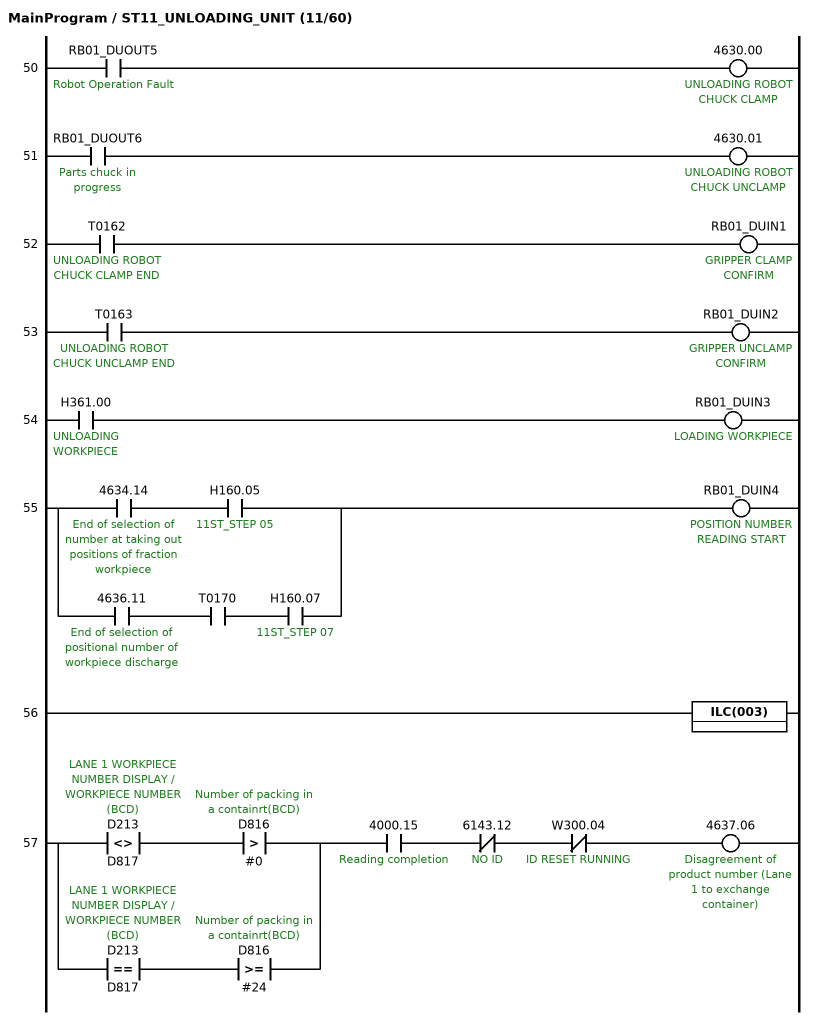
; [picture p528: MainProgram / ST11_UNLOADING_UNIT, rungs 50-57]
; rung 50
LD RB01_DUOUT5  ; Robot Operation Fault
OUT 4630.00  ; UNLOADING ROBOT CHUCK CLAMP
; rung 51
LD RB01_DUOUT6  ; Parts chuck in progress
OUT 4630.01  ; UNLOADING ROBOT CHUCK UNCLAMP
; rung 52
LD T0162  ; UNLOADING ROBOT CHUCK CLAMP END
OUT RB01_DUIN1  ; GRIPPER CLAMP CONFIRM
; rung 53
LD T0163  ; UNLOADING ROBOT CHUCK UNCLAMP END
OUT RB01_DUIN2  ; GRIPPER UNCLAMP CONFIRM
; rung 54
LD H361.00  ; UNLOADING WORKPIECE
OUT RB01_DUIN3  ; LOADING WORKPIECE
; rung 55
LD 4634.14  ; End of selection of number at taking out positions of fraction workpiece
AND H160.05  ; 11ST_STEP 05
LD 4636.11  ; End of selection of positional number of workpiece discharge
AND T0170
AND H160.07  ; 11ST_STEP 07
ORLD
OUT RB01_DUIN4  ; POSITION NUMBER READING START
; rung 56
ILC(003)
; rung 57
LD<>(305) D213 D817  ; LANE 1 WORKPIECE NUMBER DISPLAY, WORKPIECE NUMBER (BCD)
AND>(320) D816 #0  ; Number of packing in a containrt(BCD)
LD=(300) D213 D817  ; LANE 1 WORKPIECE NUMBER DISPLAY, WORKPIECE NUMBER (BCD)
AND>=(325) D816 #24  ; Number of packing in a containrt(BCD)
ORLD
AND 4000.15  ; Reading completion
ANDNOT 6143.12  ; NO ID
ANDNOT W300.04  ; ID RESET RUNNING
OUT 4637.06  ; Disagreement of product number (Lane 1 to exchange container)

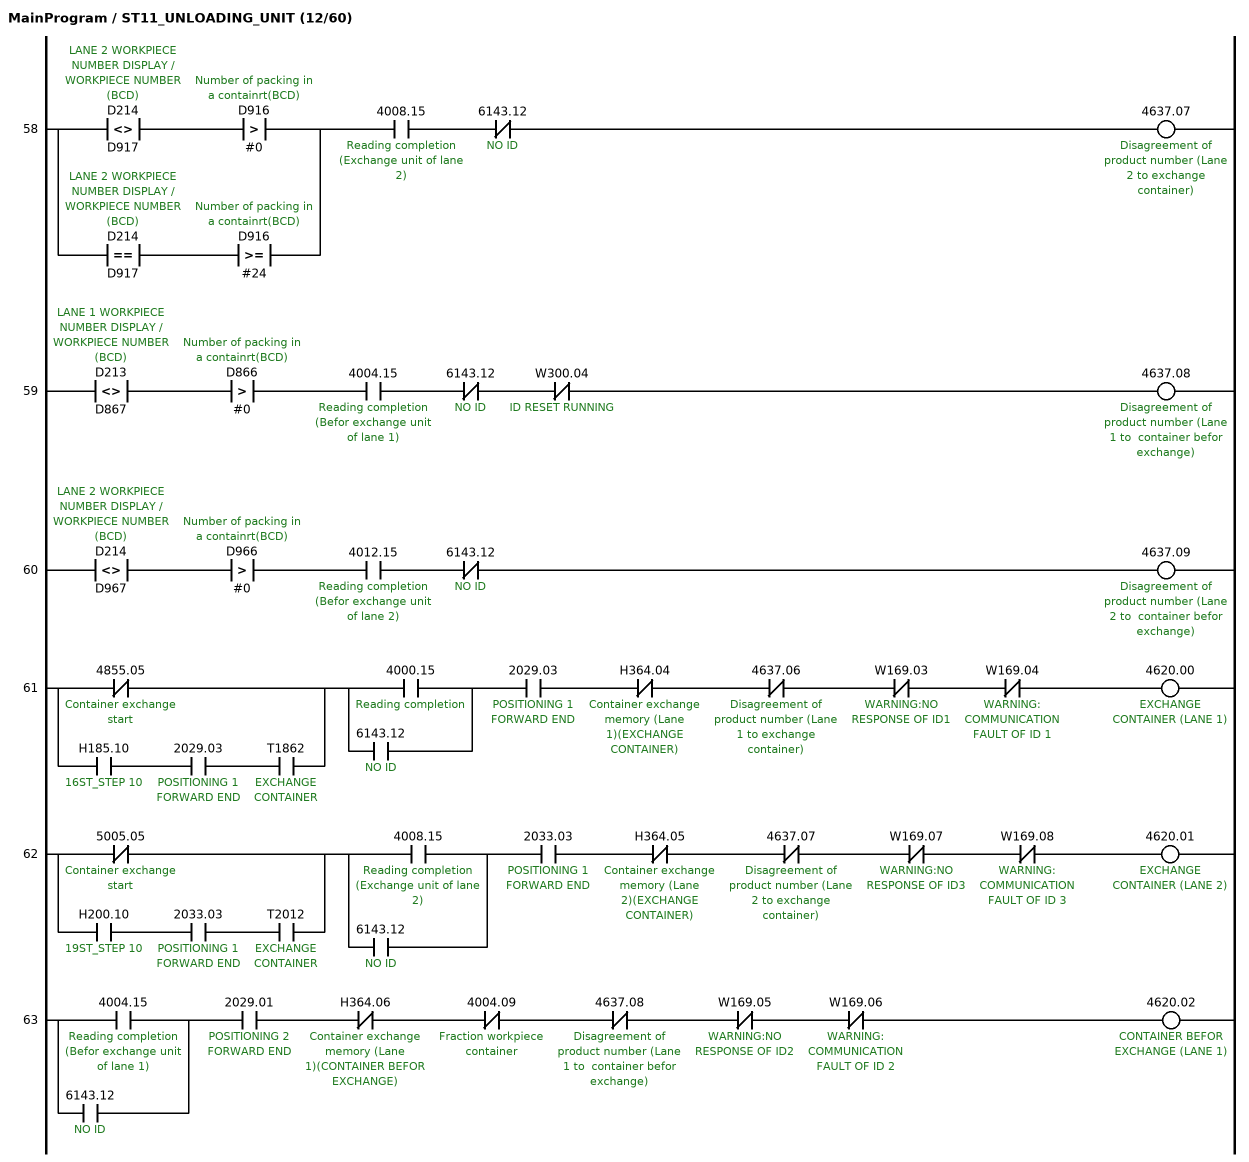
; rung 58
LD<>(305) D214 D917  ; LANE 2 WORKPIECE NUMBER DISPLAY, WORKPIECE NUMBER (BCD)
AND>(320) D916 #0  ; Number of packing in a containrt(BCD)
LD=(300) D214 D917  ; LANE 2 WORKPIECE NUMBER DISPLAY, WORKPIECE NUMBER (BCD)
AND>=(325) D916 #24  ; Number of packing in a containrt(BCD)
ORLD
AND 4008.15  ; Reading completion (Exchange unit of lane 2)
ANDNOT 6143.12  ; NO ID
OUT 4637.07  ; Disagreement of product number (Lane 2 to exchange container)
; rung 59
LD<>(305) D213 D867  ; LANE 1 WORKPIECE NUMBER DISPLAY, WORKPIECE NUMBER (BCD)
AND>(320) D866 #0  ; Number of packing in a containrt(BCD)
AND 4004.15  ; Reading completion (Befor exchange unit of lane 1)
ANDNOT 6143.12  ; NO ID
ANDNOT W300.04  ; ID RESET RUNNING
OUT 4637.08  ; Disagreement of product number (Lane 1 to  container befor exchange)
; rung 60
LD<>(305) D214 D967  ; LANE 2 WORKPIECE NUMBER DISPLAY, WORKPIECE NUMBER (BCD)
AND>(320) D966 #0  ; Number of packing in a containrt(BCD)
AND 4012.15  ; Reading completion (Befor exchange unit of lane 2)
ANDNOT 6143.12  ; NO ID
OUT 4637.09  ; Disagreement of product number (Lane 2 to  container befor exchange)
; rung 61
LDNOT 4855.05  ; Container exchange start
LD H185.10  ; 16ST_STEP 10
AND 2029.03  ; POSITIONING 1 FORWARD END
AND T1862  ; EXCHANGE CONTAINER
ORLD
LD 4000.15  ; Reading completion
OR 6143.12  ; NO ID
ANDLD
AND 2029.03  ; POSITIONING 1 FORWARD END
ANDNOT H364.04  ; Container exchange memory (Lane 1)(EXCHANGE CONTAINER)
ANDNOT 4637.06  ; Disagreement of product number (Lane 1 to exchange container)
ANDNOT W169.03  ; WARNING:NO RESPONSE OF ID1
ANDNOT W169.04  ; WARNING:COMMUNICATION FAULT OF ID 1
OUT 4620.00  ; EXCHANGE CONTAINER (LANE 1)
; rung 62
LDNOT 5005.05  ; Container exchange start
LD H200.10  ; 19ST_STEP 10
AND 2033.03  ; POSITIONING 1 FORWARD END
AND T2012  ; EXCHANGE CONTAINER
ORLD
LD 4008.15  ; Reading completion (Exchange unit of lane 2)
OR 6143.12  ; NO ID
ANDLD
AND 2033.03  ; POSITIONING 1 FORWARD END
ANDNOT H364.05  ; Container exchange memory (Lane 2)(EXCHANGE CONTAINER)
ANDNOT 4637.07  ; Disagreement of product number (Lane 2 to exchange container)
ANDNOT W169.07  ; WARNING:NO RESPONSE OF ID3
ANDNOT W169.08  ; WARNING:COMMUNICATION FAULT OF ID 3
OUT 4620.01  ; EXCHANGE CONTAINER (LANE 2)
; rung 63
LD 4004.15  ; Reading completion (Befor exchange unit of lane 1)
OR 6143.12  ; NO ID
AND 2029.01  ; POSITIONING 2 FORWARD END
ANDNOT H364.06  ; Container exchange memory (Lane 1)(CONTAINER BEFOR EXCHANGE)
ANDNOT 4004.09  ; Fraction workpiece container
ANDNOT 4637.08  ; Disagreement of product number (Lane 1 to  container befor exchange)
ANDNOT W169.05  ; WARNING:NO RESPONSE OF ID2
ANDNOT W169.06  ; WARNING:COMMUNICATION FAULT OF ID 2
OUT 4620.02  ; CONTAINER BEFOR EXCHANGE (LANE 1)

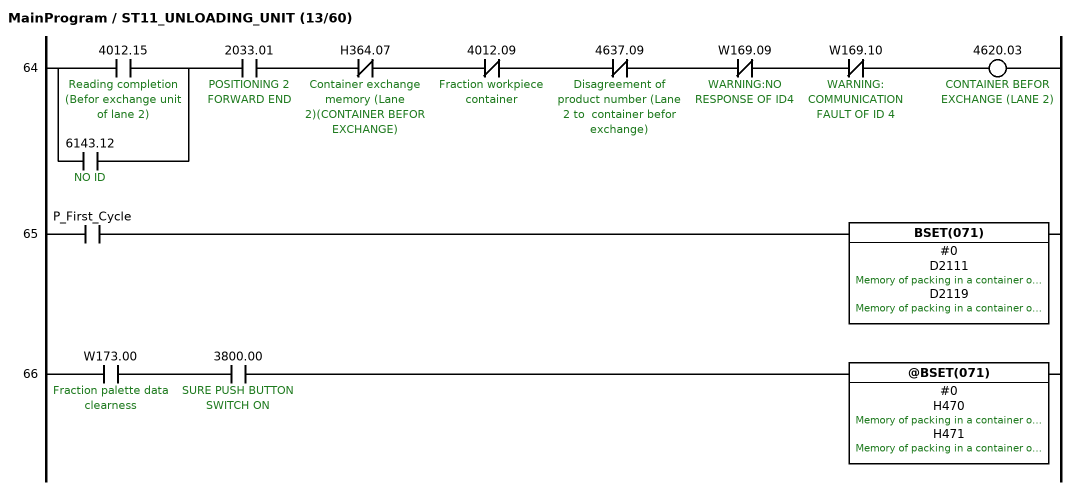
; rung 64
LD 4012.15  ; Reading completion (Befor exchange unit of lane 2)
OR 6143.12  ; NO ID
AND 2033.01  ; POSITIONING 2 FORWARD END
ANDNOT H364.07  ; Container exchange memory (Lane 2)(CONTAINER BEFOR EXCHANGE)
ANDNOT 4012.09  ; Fraction workpiece container
ANDNOT 4637.09  ; Disagreement of product number (Lane 2 to  container befor exchange)
ANDNOT W169.09  ; WARNING:NO RESPONSE OF ID4
ANDNOT W169.10  ; WARNING:COMMUNICATION FAULT OF ID 4
OUT 4620.03  ; CONTAINER BEFOR EXCHANGE (LANE 2)
; rung 65
LD P_First_Cycle
BSET(071) #0 D2111 D2119  ; Memory of packing in a container of fraction workpiece (code no.1), Memory of packing in a container of fraction workpiece (code no.9)
; rung 66
LD W173.00  ; Fraction palette data clearness
AND 3800.00  ; SURE PUSH BUTTON SWITCH ON
@BSET(071) #0 H470 H471  ; Memory of packing in a container of fraction workpiece

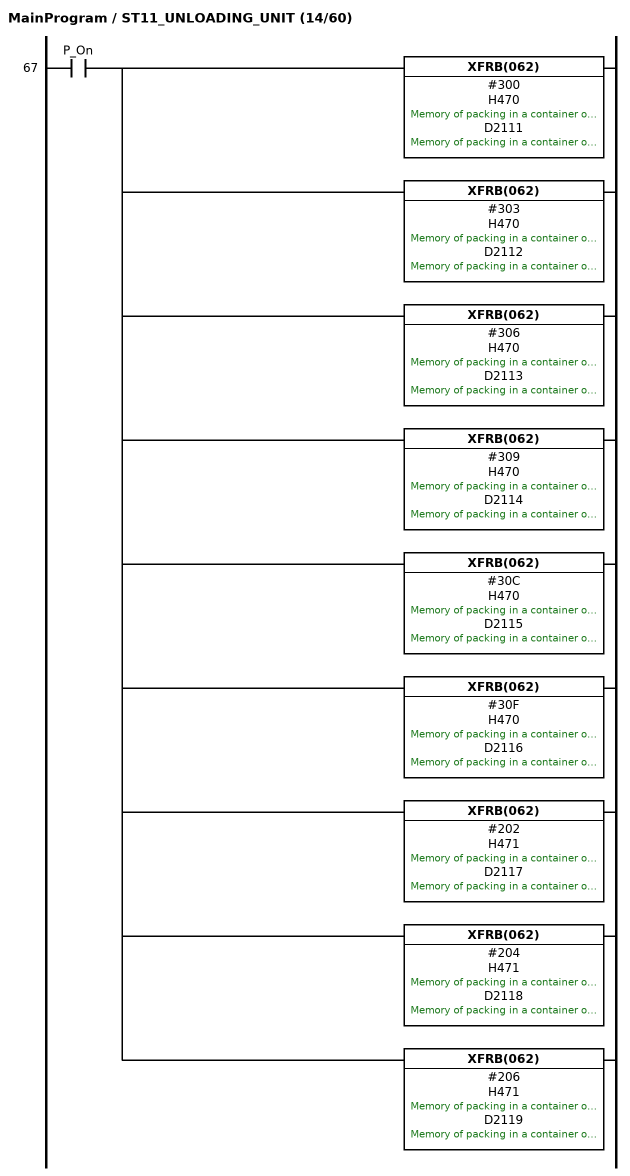
; rung 67
LD P_On
XFRB(062) #300 H470 D2111  ; Memory of packing in a container of fraction workpiece, Memory of packing in a container of fraction workpiece (code no.1)
XFRB(062) #303 H470 D2112  ; Memory of packing in a container of fraction workpiece, Memory of packing in a container of fraction workpiece (code no.2)
XFRB(062) #306 H470 D2113  ; Memory of packing in a container of fraction workpiece, Memory of packing in a container of fraction workpiece (code no.3)
XFRB(062) #309 H470 D2114  ; Memory of packing in a container of fraction workpiece, Memory of packing in a container of fraction workpiece (code no.4)
XFRB(062) #30C H470 D2115  ; Memory of packing in a container of fraction workpiece, Memory of packing in a container of fraction workpiece (code no.5)
XFRB(062) #30F H470 D2116  ; Memory of packing in a container of fraction workpiece, Memory of packing in a container of fraction workpiece (code no.6)
XFRB(062) #202 H471 D2117  ; Memory of packing in a container of fraction workpiece, Memory of packing in a container of fraction workpiece (code no.7)
XFRB(062) #204 H471 D2118  ; Memory of packing in a container of fraction workpiece, Memory of packing in a container of fraction workpiece (code no.8)
XFRB(062) #206 H471 D2119  ; Memory of packing in a container of fraction workpiece, Memory of packing in a container of fraction workpiece (code no.9)

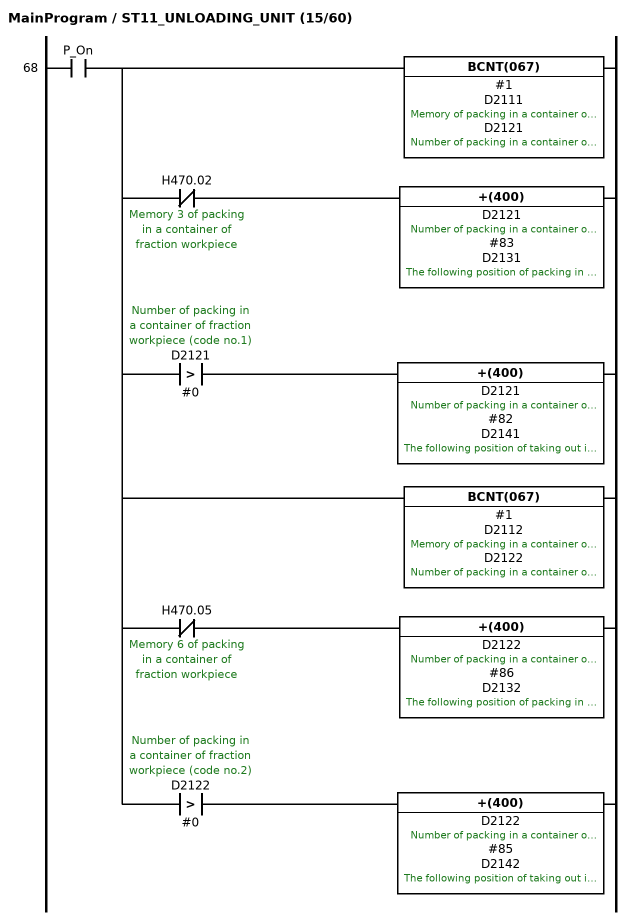
; rung 68
LD P_On
OUT TR0
BCNT(067) #1 D2111 D2121  ; Memory of packing in a container of fraction workpiece (code no.1), Number of packing in a container of fraction workpiece (code no.1)
ANDNOT H470.02  ; Memory 3 of packing in a container of fraction workpiece
+(400) D2121 #83 D2131  ; Number of packing in a container of fraction workpiece (code no.1), The following position of packing in a container number in fraction workpiece (code no.1)
LD TR0
AND>(320) D2121 #0  ; Number of packing in a container of fraction workpiece (code no.1)
+(400) D2121 #82 D2141  ; Number of packing in a container of fraction workpiece (code no.1), The following position of taking out in a container number in fraction workpiece (code no.1)
LD TR0
BCNT(067) #1 D2112 D2122  ; Memory of packing in a container of fraction workpiece (code no.2), Number of packing in a container of fraction workpiece (code no.2)
ANDNOT H470.05  ; Memory 6 of packing in a container of fraction workpiece
+(400) D2122 #86 D2132  ; Number of packing in a container of fraction workpiece (code no.2), The following position of packing in a container number in fraction workpiece (code no.2)
LD TR0
AND>(320) D2122 #0  ; Number of packing in a container of fraction workpiece (code no.2)
+(400) D2122 #85 D2142  ; Number of packing in a container of fraction workpiece (code no.2), The following position of taking out in a container number in fraction workpiece (code no.2)

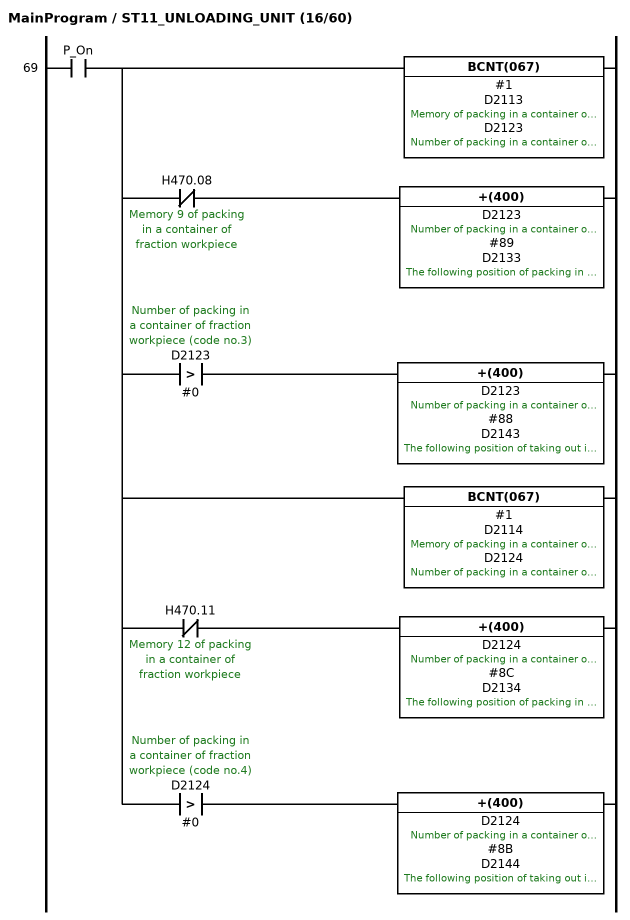
; rung 69
LD P_On
OUT TR0
BCNT(067) #1 D2113 D2123  ; Memory of packing in a container of fraction workpiece (code no.3), Number of packing in a container of fraction workpiece (code no.3)
ANDNOT H470.08  ; Memory 9 of packing in a container of fraction workpiece
+(400) D2123 #89 D2133  ; Number of packing in a container of fraction workpiece (code no.3), The following position of packing in a container number in fraction workpiece (code no.3)
LD TR0
AND>(320) D2123 #0  ; Number of packing in a container of fraction workpiece (code no.3)
+(400) D2123 #88 D2143  ; Number of packing in a container of fraction workpiece (code no.3), The following position of taking out in a container number in fraction workpiece (code no.3)
LD TR0
BCNT(067) #1 D2114 D2124  ; Memory of packing in a container of fraction workpiece (code no.4), Number of packing in a container of fraction workpiece (code no.4)
ANDNOT H470.11  ; Memory 12 of packing in a container of fraction workpiece
+(400) D2124 #8C D2134  ; Number of packing in a container of fraction workpiece (code no.4), The following position of packing in a container number in fraction workpiece (code no.4)
LD TR0
AND>(320) D2124 #0  ; Number of packing in a container of fraction workpiece (code no.4)
+(400) D2124 #8B D2144  ; Number of packing in a container of fraction workpiece (code no.4), The following position of taking out in a container number in fraction workpiece (code no.4)

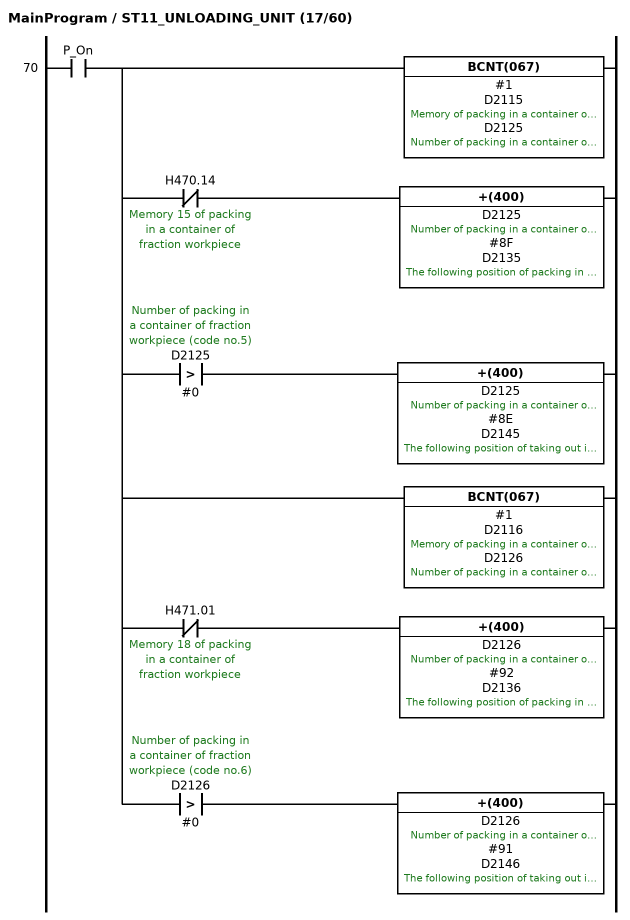
; rung 70
LD P_On
OUT TR0
BCNT(067) #1 D2115 D2125  ; Memory of packing in a container of fraction workpiece (code no.5), Number of packing in a container of fraction workpiece (code no.5)
ANDNOT H470.14  ; Memory 15 of packing in a container of fraction workpiece
+(400) D2125 #8F D2135  ; Number of packing in a container of fraction workpiece (code no.5), The following position of packing in a container number in fraction workpiece (code no.5)
LD TR0
AND>(320) D2125 #0  ; Number of packing in a container of fraction workpiece (code no.5)
+(400) D2125 #8E D2145  ; Number of packing in a container of fraction workpiece (code no.5), The following position of taking out in a container number in fraction workpiece (code no.5)
LD TR0
BCNT(067) #1 D2116 D2126  ; Memory of packing in a container of fraction workpiece (code no.6), Number of packing in a container of fraction workpiece (code no.6)
ANDNOT H471.01  ; Memory 18 of packing in a container of fraction workpiece
+(400) D2126 #92 D2136  ; Number of packing in a container of fraction workpiece (code no.6), The following position of packing in a container number in fraction workpiece (code no.6)
LD TR0
AND>(320) D2126 #0  ; Number of packing in a container of fraction workpiece (code no.6)
+(400) D2126 #91 D2146  ; Number of packing in a container of fraction workpiece (code no.6), The following position of taking out in a container number in fraction workpiece (code no.6)

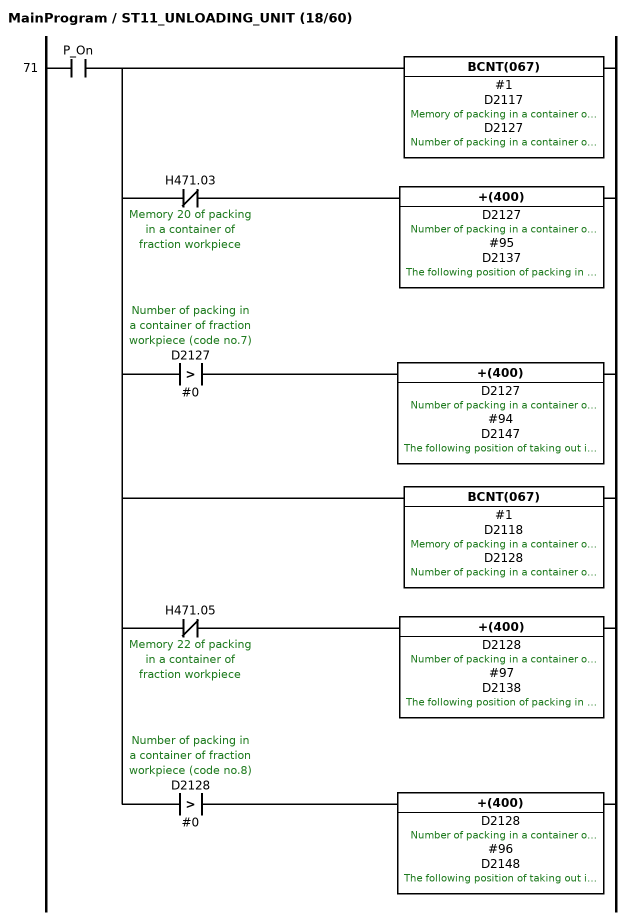
; rung 71
LD P_On
OUT TR0
BCNT(067) #1 D2117 D2127  ; Memory of packing in a container of fraction workpiece (code no.7), Number of packing in a container of fraction workpiece (code no.7)
ANDNOT H471.03  ; Memory 20 of packing in a container of fraction workpiece
+(400) D2127 #95 D2137  ; Number of packing in a container of fraction workpiece (code no.7), The following position of packing in a container number in fraction workpiece (code no.7)
LD TR0
AND>(320) D2127 #0  ; Number of packing in a container of fraction workpiece (code no.7)
+(400) D2127 #94 D2147  ; Number of packing in a container of fraction workpiece (code no.7), The following position of taking out in a container number in fraction workpiece (code no.7)
LD TR0
BCNT(067) #1 D2118 D2128  ; Memory of packing in a container of fraction workpiece (code no.8), Number of packing in a container of fraction workpiece (code no.8)
ANDNOT H471.05  ; Memory 22 of packing in a container of fraction workpiece
+(400) D2128 #97 D2138  ; Number of packing in a container of fraction workpiece (code no.8), The following position of packing in a container number in fraction workpiece (code no.8)
LD TR0
AND>(320) D2128 #0  ; Number of packing in a container of fraction workpiece (code no.8)
+(400) D2128 #96 D2148  ; Number of packing in a container of fraction workpiece (code no.8), The following position of taking out in a container number in fraction workpiece (code no.8)

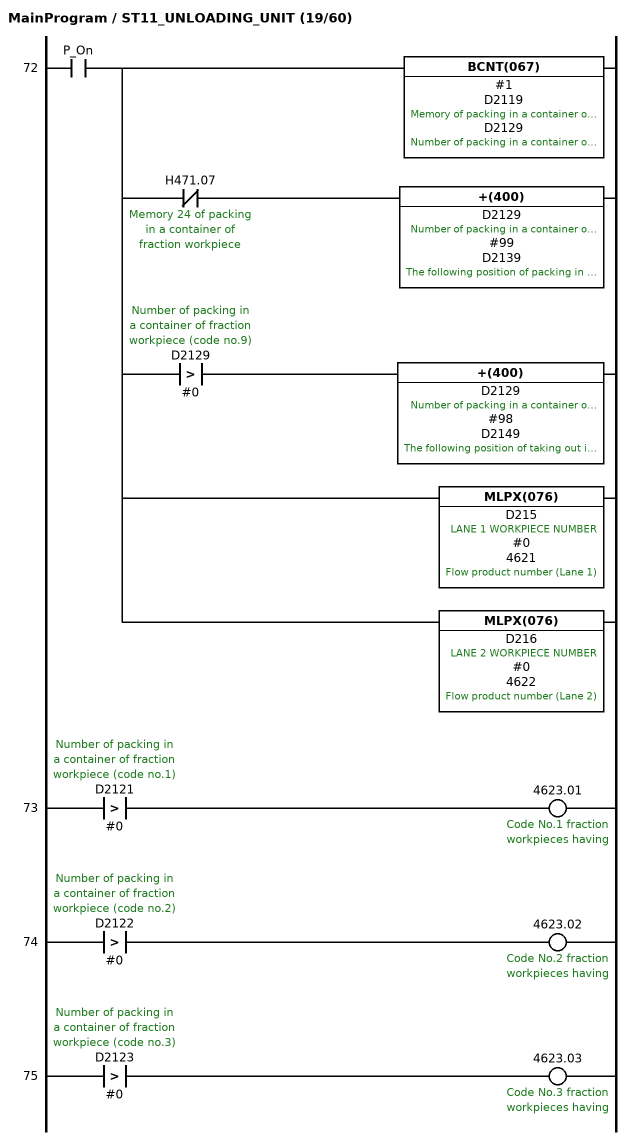
; rung 72
LD P_On
OUT TR0
BCNT(067) #1 D2119 D2129  ; Memory of packing in a container of fraction workpiece (code no.9), Number of packing in a container of fraction workpiece (code no.9)
ANDNOT H471.07  ; Memory 24 of packing in a container of fraction workpiece
+(400) D2129 #99 D2139  ; Number of packing in a container of fraction workpiece (code no.9), The following position of packing in a container number in fraction workpiece (code no.9)
LD TR0
AND>(320) D2129 #0  ; Number of packing in a container of fraction workpiece (code no.9)
+(400) D2129 #98 D2149  ; Number of packing in a container of fraction workpiece (code no.9), The following position of taking out in a container number in fraction workpiece (code no.9)
LD TR0
MLPX(076) D215 #0 4621  ; LANE 1 WORKPIECE NUMBER, Flow product number (Lane 1)
MLPX(076) D216 #0 4622  ; LANE 2 WORKPIECE NUMBER, Flow product number (Lane 2)
; rung 73
LD>(320) D2121 #0  ; Number of packing in a container of fraction workpiece (code no.1)
OUT 4623.01  ; Code No.1 fraction workpieces having
; rung 74
LD>(320) D2122 #0  ; Number of packing in a container of fraction workpiece (code no.2)
OUT 4623.02  ; Code No.2 fraction workpieces having
; rung 75
LD>(320) D2123 #0  ; Number of packing in a container of fraction workpiece (code no.3)
OUT 4623.03  ; Code No.3 fraction workpieces having

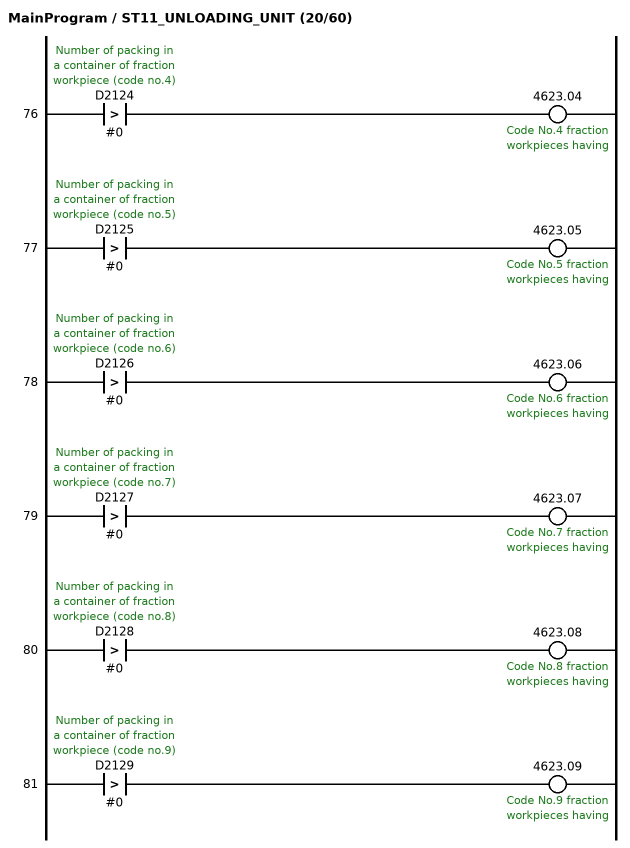
; rung 76
LD>(320) D2124 #0  ; Number of packing in a container of fraction workpiece (code no.4)
OUT 4623.04  ; Code No.4 fraction workpieces having
; rung 77
LD>(320) D2125 #0  ; Number of packing in a container of fraction workpiece (code no.5)
OUT 4623.05  ; Code No.5 fraction workpieces having
; rung 78
LD>(320) D2126 #0  ; Number of packing in a container of fraction workpiece (code no.6)
OUT 4623.06  ; Code No.6 fraction workpieces having
; rung 79
LD>(320) D2127 #0  ; Number of packing in a container of fraction workpiece (code no.7)
OUT 4623.07  ; Code No.7 fraction workpieces having
; rung 80
LD>(320) D2128 #0  ; Number of packing in a container of fraction workpiece (code no.8)
OUT 4623.08  ; Code No.8 fraction workpieces having
; rung 81
LD>(320) D2129 #0  ; Number of packing in a container of fraction workpiece (code no.9)
OUT 4623.09  ; Code No.9 fraction workpieces having

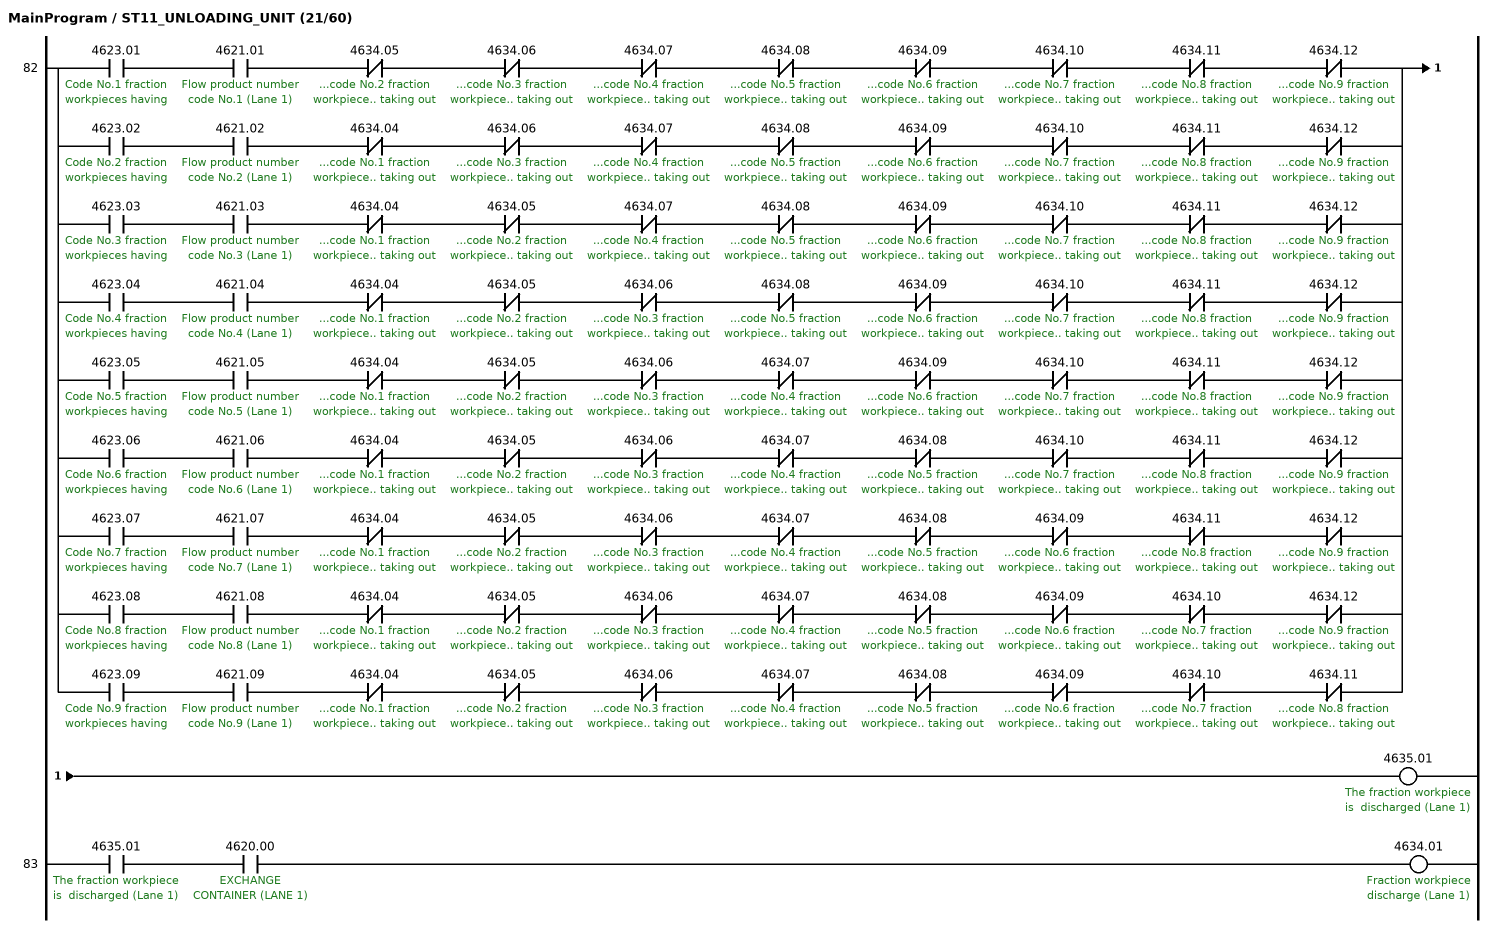
; rung 82
LD 4623.01  ; Code No.1 fraction workpieces having
AND 4621.01  ; Flow product number code No.1 (Lane 1)
ANDNOT 4634.05  ; ...code No.2 fraction workpiece.. taking out
ANDNOT 4634.06  ; ...code No.3 fraction workpiece.. taking out
ANDNOT 4634.07  ; ...code No.4 fraction workpiece.. taking out
ANDNOT 4634.08  ; ...code No.5 fraction workpiece.. taking out
ANDNOT 4634.09  ; ...code No.6 fraction workpiece.. taking out
ANDNOT 4634.10  ; ...code No.7 fraction workpiece.. taking out
ANDNOT 4634.11  ; ...code No.8 fraction workpiece.. taking out
ANDNOT 4634.12  ; ...code No.9 fraction workpiece.. taking out
LD 4623.02  ; Code No.2 fraction workpieces having
AND 4621.02  ; Flow product number code No.2 (Lane 1)
ANDNOT 4634.04  ; ...code No.1 fraction workpiece.. taking out
ANDNOT 4634.06  ; ...code No.3 fraction workpiece.. taking out
ANDNOT 4634.07  ; ...code No.4 fraction workpiece.. taking out
ANDNOT 4634.08  ; ...code No.5 fraction workpiece.. taking out
ANDNOT 4634.09  ; ...code No.6 fraction workpiece.. taking out
ANDNOT 4634.10  ; ...code No.7 fraction workpiece.. taking out
ANDNOT 4634.11  ; ...code No.8 fraction workpiece.. taking out
ANDNOT 4634.12  ; ...code No.9 fraction workpiece.. taking out
ORLD
LD 4623.03  ; Code No.3 fraction workpieces having
AND 4621.03  ; Flow product number code No.3 (Lane 1)
ANDNOT 4634.04  ; ...code No.1 fraction workpiece.. taking out
ANDNOT 4634.05  ; ...code No.2 fraction workpiece.. taking out
ANDNOT 4634.07  ; ...code No.4 fraction workpiece.. taking out
ANDNOT 4634.08  ; ...code No.5 fraction workpiece.. taking out
ANDNOT 4634.09  ; ...code No.6 fraction workpiece.. taking out
ANDNOT 4634.10  ; ...code No.7 fraction workpiece.. taking out
ANDNOT 4634.11  ; ...code No.8 fraction workpiece.. taking out
ANDNOT 4634.12  ; ...code No.9 fraction workpiece.. taking out
ORLD
LD 4623.04  ; Code No.4 fraction workpieces having
AND 4621.04  ; Flow product number code No.4 (Lane 1)
ANDNOT 4634.04  ; ...code No.1 fraction workpiece.. taking out
ANDNOT 4634.05  ; ...code No.2 fraction workpiece.. taking out
ANDNOT 4634.06  ; ...code No.3 fraction workpiece.. taking out
ANDNOT 4634.08  ; ...code No.5 fraction workpiece.. taking out
ANDNOT 4634.09  ; ...code No.6 fraction workpiece.. taking out
ANDNOT 4634.10  ; ...code No.7 fraction workpiece.. taking out
ANDNOT 4634.11  ; ...code No.8 fraction workpiece.. taking out
ANDNOT 4634.12  ; ...code No.9 fraction workpiece.. taking out
ORLD
LD 4623.05  ; Code No.5 fraction workpieces having
AND 4621.05  ; Flow product number code No.5 (Lane 1)
ANDNOT 4634.04  ; ...code No.1 fraction workpiece.. taking out
ANDNOT 4634.05  ; ...code No.2 fraction workpiece.. taking out
ANDNOT 4634.06  ; ...code No.3 fraction workpiece.. taking out
ANDNOT 4634.07  ; ...code No.4 fraction workpiece.. taking out
ANDNOT 4634.09  ; ...code No.6 fraction workpiece.. taking out
ANDNOT 4634.10  ; ...code No.7 fraction workpiece.. taking out
ANDNOT 4634.11  ; ...code No.8 fraction workpiece.. taking out
ANDNOT 4634.12  ; ...code No.9 fraction workpiece.. taking out
ORLD
LD 4623.06  ; Code No.6 fraction workpieces having
AND 4621.06  ; Flow product number code No.6 (Lane 1)
ANDNOT 4634.04  ; ...code No.1 fraction workpiece.. taking out
ANDNOT 4634.05  ; ...code No.2 fraction workpiece.. taking out
ANDNOT 4634.06  ; ...code No.3 fraction workpiece.. taking out
ANDNOT 4634.07  ; ...code No.4 fraction workpiece.. taking out
ANDNOT 4634.08  ; ...code No.5 fraction workpiece.. taking out
ANDNOT 4634.10  ; ...code No.7 fraction workpiece.. taking out
ANDNOT 4634.11  ; ...code No.8 fraction workpiece.. taking out
ANDNOT 4634.12  ; ...code No.9 fraction workpiece.. taking out
ORLD
LD 4623.07  ; Code No.7 fraction workpieces having
AND 4621.07  ; Flow product number code No.7 (Lane 1)
ANDNOT 4634.04  ; ...code No.1 fraction workpiece.. taking out
ANDNOT 4634.05  ; ...code No.2 fraction workpiece.. taking out
ANDNOT 4634.06  ; ...code No.3 fraction workpiece.. taking out
ANDNOT 4634.07  ; ...code No.4 fraction workpiece.. taking out
ANDNOT 4634.08  ; ...code No.5 fraction workpiece.. taking out
ANDNOT 4634.09  ; ...code No.6 fraction workpiece.. taking out
ANDNOT 4634.11  ; ...code No.8 fraction workpiece.. taking out
ANDNOT 4634.12  ; ...code No.9 fraction workpiece.. taking out
ORLD
LD 4623.08  ; Code No.8 fraction workpieces having
AND 4621.08  ; Flow product number code No.8 (Lane 1)
ANDNOT 4634.04  ; ...code No.1 fraction workpiece.. taking out
ANDNOT 4634.05  ; ...code No.2 fraction workpiece.. taking out
ANDNOT 4634.06  ; ...code No.3 fraction workpiece.. taking out
ANDNOT 4634.07  ; ...code No.4 fraction workpiece.. taking out
ANDNOT 4634.08  ; ...code No.5 fraction workpiece.. taking out
ANDNOT 4634.09  ; ...code No.6 fraction workpiece.. taking out
ANDNOT 4634.10  ; ...code No.7 fraction workpiece.. taking out
ANDNOT 4634.12  ; ...code No.9 fraction workpiece.. taking out
ORLD
LD 4623.09  ; Code No.9 fraction workpieces having
AND 4621.09  ; Flow product number code No.9 (Lane 1)
ANDNOT 4634.04  ; ...code No.1 fraction workpiece.. taking out
ANDNOT 4634.05  ; ...code No.2 fraction workpiece.. taking out
ANDNOT 4634.06  ; ...code No.3 fraction workpiece.. taking out
ANDNOT 4634.07  ; ...code No.4 fraction workpiece.. taking out
ANDNOT 4634.08  ; ...code No.5 fraction workpiece.. taking out
ANDNOT 4634.09  ; ...code No.6 fraction workpiece.. taking out
ANDNOT 4634.10  ; ...code No.7 fraction workpiece.. taking out
ANDNOT 4634.11  ; ...code No.8 fraction workpiece.. taking out
ORLD
OUT 4635.01  ; The fraction workpiece is  discharged (Lane 1)
; rung 83
LD 4635.01  ; The fraction workpiece is  discharged (Lane 1)
AND 4620.00  ; EXCHANGE CONTAINER (LANE 1)
OUT 4634.01  ; Fraction workpiece discharge (Lane 1)

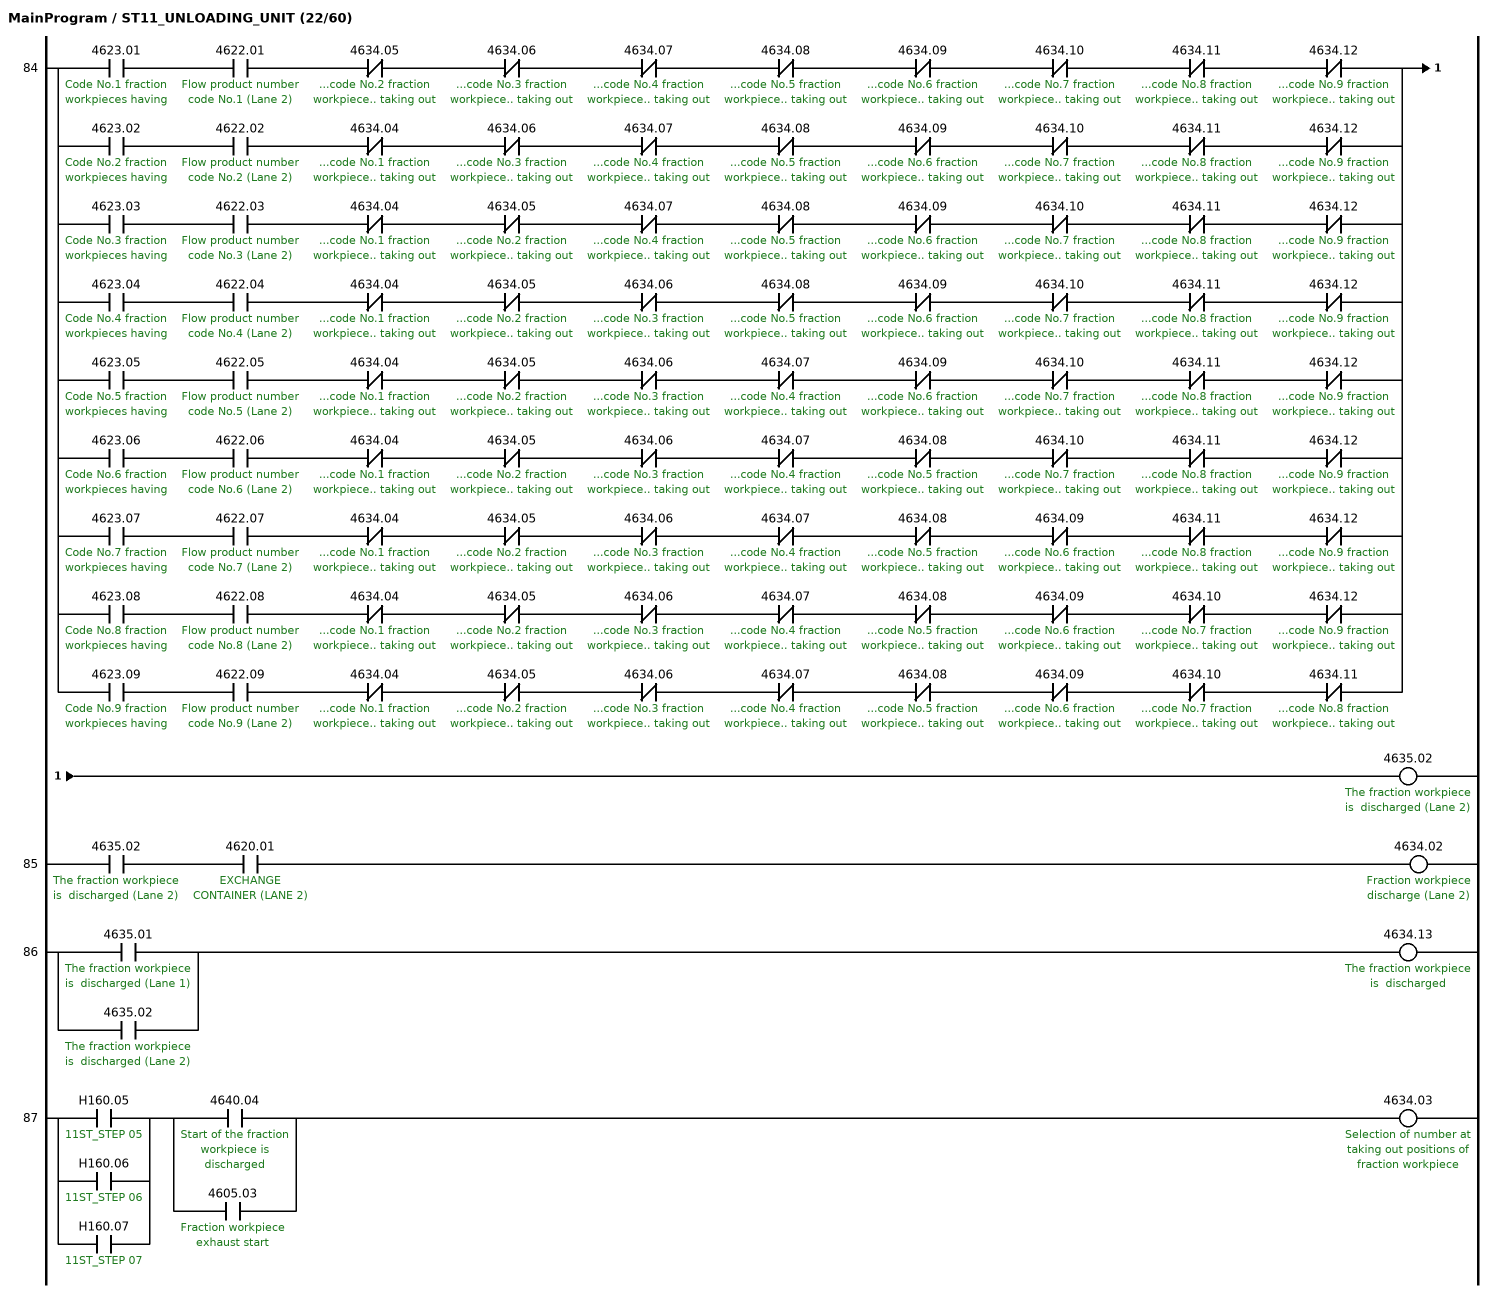
; rung 84
LD 4623.01  ; Code No.1 fraction workpieces having
AND 4622.01  ; Flow product number code No.1 (Lane 2)
ANDNOT 4634.05  ; ...code No.2 fraction workpiece.. taking out
ANDNOT 4634.06  ; ...code No.3 fraction workpiece.. taking out
ANDNOT 4634.07  ; ...code No.4 fraction workpiece.. taking out
ANDNOT 4634.08  ; ...code No.5 fraction workpiece.. taking out
ANDNOT 4634.09  ; ...code No.6 fraction workpiece.. taking out
ANDNOT 4634.10  ; ...code No.7 fraction workpiece.. taking out
ANDNOT 4634.11  ; ...code No.8 fraction workpiece.. taking out
ANDNOT 4634.12  ; ...code No.9 fraction workpiece.. taking out
LD 4623.02  ; Code No.2 fraction workpieces having
AND 4622.02  ; Flow product number code No.2 (Lane 2)
ANDNOT 4634.04  ; ...code No.1 fraction workpiece.. taking out
ANDNOT 4634.06  ; ...code No.3 fraction workpiece.. taking out
ANDNOT 4634.07  ; ...code No.4 fraction workpiece.. taking out
ANDNOT 4634.08  ; ...code No.5 fraction workpiece.. taking out
ANDNOT 4634.09  ; ...code No.6 fraction workpiece.. taking out
ANDNOT 4634.10  ; ...code No.7 fraction workpiece.. taking out
ANDNOT 4634.11  ; ...code No.8 fraction workpiece.. taking out
ANDNOT 4634.12  ; ...code No.9 fraction workpiece.. taking out
ORLD
LD 4623.03  ; Code No.3 fraction workpieces having
AND 4622.03  ; Flow product number code No.3 (Lane 2)
ANDNOT 4634.04  ; ...code No.1 fraction workpiece.. taking out
ANDNOT 4634.05  ; ...code No.2 fraction workpiece.. taking out
ANDNOT 4634.07  ; ...code No.4 fraction workpiece.. taking out
ANDNOT 4634.08  ; ...code No.5 fraction workpiece.. taking out
ANDNOT 4634.09  ; ...code No.6 fraction workpiece.. taking out
ANDNOT 4634.10  ; ...code No.7 fraction workpiece.. taking out
ANDNOT 4634.11  ; ...code No.8 fraction workpiece.. taking out
ANDNOT 4634.12  ; ...code No.9 fraction workpiece.. taking out
ORLD
LD 4623.04  ; Code No.4 fraction workpieces having
AND 4622.04  ; Flow product number code No.4 (Lane 2)
ANDNOT 4634.04  ; ...code No.1 fraction workpiece.. taking out
ANDNOT 4634.05  ; ...code No.2 fraction workpiece.. taking out
ANDNOT 4634.06  ; ...code No.3 fraction workpiece.. taking out
ANDNOT 4634.08  ; ...code No.5 fraction workpiece.. taking out
ANDNOT 4634.09  ; ...code No.6 fraction workpiece.. taking out
ANDNOT 4634.10  ; ...code No.7 fraction workpiece.. taking out
ANDNOT 4634.11  ; ...code No.8 fraction workpiece.. taking out
ANDNOT 4634.12  ; ...code No.9 fraction workpiece.. taking out
ORLD
LD 4623.05  ; Code No.5 fraction workpieces having
AND 4622.05  ; Flow product number code No.5 (Lane 2)
ANDNOT 4634.04  ; ...code No.1 fraction workpiece.. taking out
ANDNOT 4634.05  ; ...code No.2 fraction workpiece.. taking out
ANDNOT 4634.06  ; ...code No.3 fraction workpiece.. taking out
ANDNOT 4634.07  ; ...code No.4 fraction workpiece.. taking out
ANDNOT 4634.09  ; ...code No.6 fraction workpiece.. taking out
ANDNOT 4634.10  ; ...code No.7 fraction workpiece.. taking out
ANDNOT 4634.11  ; ...code No.8 fraction workpiece.. taking out
ANDNOT 4634.12  ; ...code No.9 fraction workpiece.. taking out
ORLD
LD 4623.06  ; Code No.6 fraction workpieces having
AND 4622.06  ; Flow product number code No.6 (Lane 2)
ANDNOT 4634.04  ; ...code No.1 fraction workpiece.. taking out
ANDNOT 4634.05  ; ...code No.2 fraction workpiece.. taking out
ANDNOT 4634.06  ; ...code No.3 fraction workpiece.. taking out
ANDNOT 4634.07  ; ...code No.4 fraction workpiece.. taking out
ANDNOT 4634.08  ; ...code No.5 fraction workpiece.. taking out
ANDNOT 4634.10  ; ...code No.7 fraction workpiece.. taking out
ANDNOT 4634.11  ; ...code No.8 fraction workpiece.. taking out
ANDNOT 4634.12  ; ...code No.9 fraction workpiece.. taking out
ORLD
LD 4623.07  ; Code No.7 fraction workpieces having
AND 4622.07  ; Flow product number code No.7 (Lane 2)
ANDNOT 4634.04  ; ...code No.1 fraction workpiece.. taking out
ANDNOT 4634.05  ; ...code No.2 fraction workpiece.. taking out
ANDNOT 4634.06  ; ...code No.3 fraction workpiece.. taking out
ANDNOT 4634.07  ; ...code No.4 fraction workpiece.. taking out
ANDNOT 4634.08  ; ...code No.5 fraction workpiece.. taking out
ANDNOT 4634.09  ; ...code No.6 fraction workpiece.. taking out
ANDNOT 4634.11  ; ...code No.8 fraction workpiece.. taking out
ANDNOT 4634.12  ; ...code No.9 fraction workpiece.. taking out
ORLD
LD 4623.08  ; Code No.8 fraction workpieces having
AND 4622.08  ; Flow product number code No.8 (Lane 2)
ANDNOT 4634.04  ; ...code No.1 fraction workpiece.. taking out
ANDNOT 4634.05  ; ...code No.2 fraction workpiece.. taking out
ANDNOT 4634.06  ; ...code No.3 fraction workpiece.. taking out
ANDNOT 4634.07  ; ...code No.4 fraction workpiece.. taking out
ANDNOT 4634.08  ; ...code No.5 fraction workpiece.. taking out
ANDNOT 4634.09  ; ...code No.6 fraction workpiece.. taking out
ANDNOT 4634.10  ; ...code No.7 fraction workpiece.. taking out
ANDNOT 4634.12  ; ...code No.9 fraction workpiece.. taking out
ORLD
LD 4623.09  ; Code No.9 fraction workpieces having
AND 4622.09  ; Flow product number code No.9 (Lane 2)
ANDNOT 4634.04  ; ...code No.1 fraction workpiece.. taking out
ANDNOT 4634.05  ; ...code No.2 fraction workpiece.. taking out
ANDNOT 4634.06  ; ...code No.3 fraction workpiece.. taking out
ANDNOT 4634.07  ; ...code No.4 fraction workpiece.. taking out
ANDNOT 4634.08  ; ...code No.5 fraction workpiece.. taking out
ANDNOT 4634.09  ; ...code No.6 fraction workpiece.. taking out
ANDNOT 4634.10  ; ...code No.7 fraction workpiece.. taking out
ANDNOT 4634.11  ; ...code No.8 fraction workpiece.. taking out
ORLD
OUT 4635.02  ; The fraction workpiece is  discharged (Lane 2)
; rung 85
LD 4635.02  ; The fraction workpiece is  discharged (Lane 2)
AND 4620.01  ; EXCHANGE CONTAINER (LANE 2)
OUT 4634.02  ; Fraction workpiece discharge (Lane 2)
; rung 86
LD 4635.01  ; The fraction workpiece is  discharged (Lane 1)
OR 4635.02  ; The fraction workpiece is  discharged (Lane 2)
OUT 4634.13  ; The fraction workpiece is  discharged
; rung 87
LD H160.05  ; 11ST_STEP 05
OR H160.06  ; 11ST_STEP 06
OR H160.07  ; 11ST_STEP 07
LD 4640.04  ; Start of the fraction workpiece is discharged
OR 4605.03  ; Fraction workpiece exhaust start
ANDLD
OUT 4634.03  ; Selection of number at taking out positions of fraction workpiece

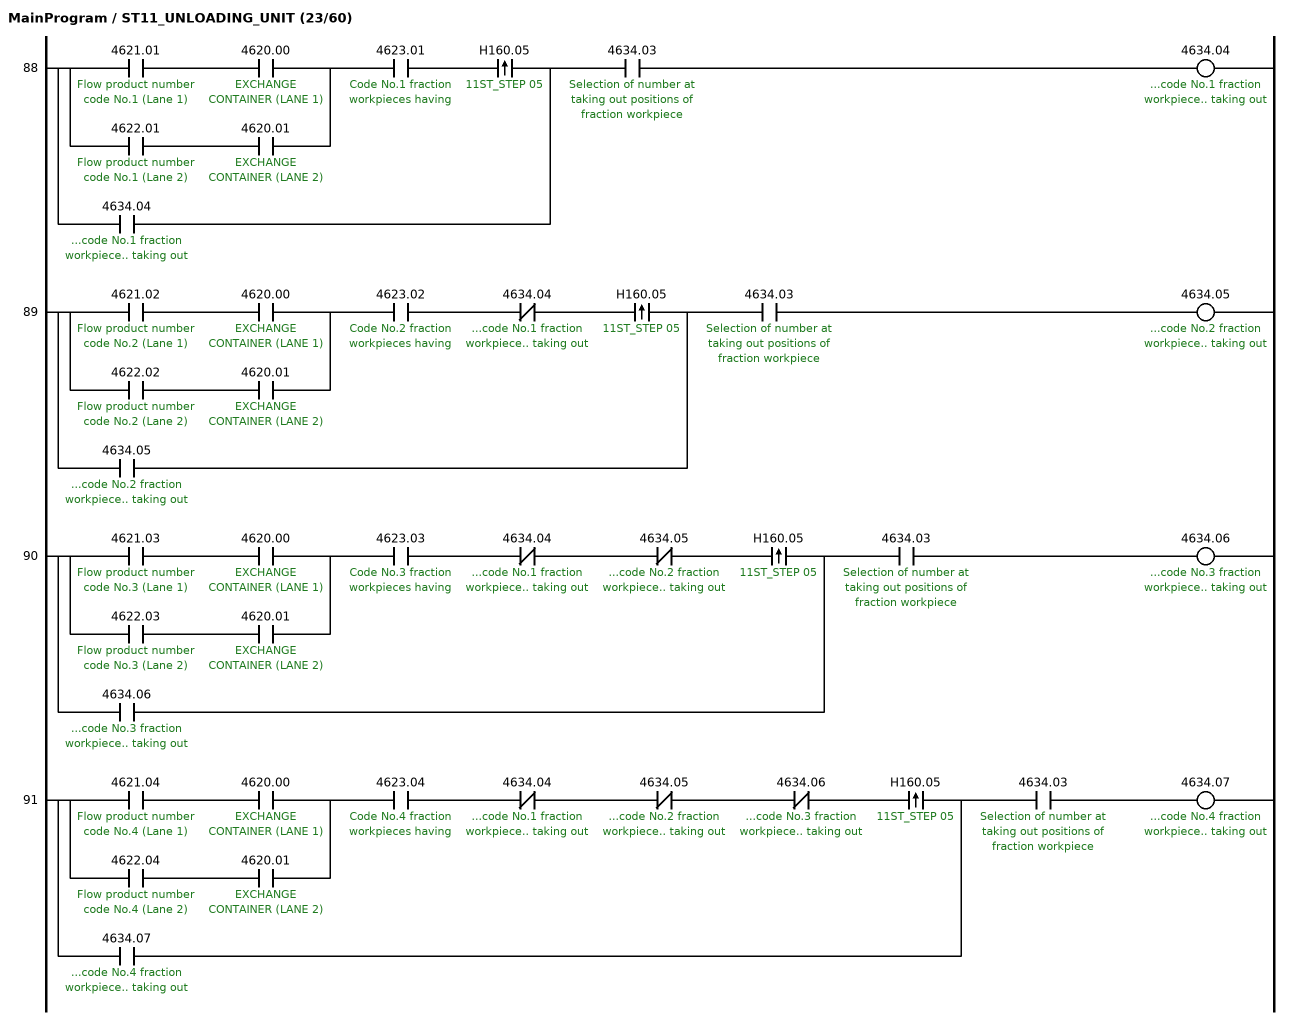
; rung 88
LD 4621.01  ; Flow product number code No.1 (Lane 1)
AND 4620.00  ; EXCHANGE CONTAINER (LANE 1)
LD 4622.01  ; Flow product number code No.1 (Lane 2)
AND 4620.01  ; EXCHANGE CONTAINER (LANE 2)
ORLD
AND 4623.01  ; Code No.1 fraction workpieces having
@AND H160.05  ; 11ST_STEP 05
OR 4634.04  ; ...code No.1 fraction workpiece.. taking out
AND 4634.03  ; Selection of number at taking out positions of fraction workpiece
OUT 4634.04  ; ...code No.1 fraction workpiece.. taking out
; rung 89
LD 4621.02  ; Flow product number code No.2 (Lane 1)
AND 4620.00  ; EXCHANGE CONTAINER (LANE 1)
LD 4622.02  ; Flow product number code No.2 (Lane 2)
AND 4620.01  ; EXCHANGE CONTAINER (LANE 2)
ORLD
AND 4623.02  ; Code No.2 fraction workpieces having
ANDNOT 4634.04  ; ...code No.1 fraction workpiece.. taking out
@AND H160.05  ; 11ST_STEP 05
OR 4634.05  ; ...code No.2 fraction workpiece.. taking out
AND 4634.03  ; Selection of number at taking out positions of fraction workpiece
OUT 4634.05  ; ...code No.2 fraction workpiece.. taking out
; rung 90
LD 4621.03  ; Flow product number code No.3 (Lane 1)
AND 4620.00  ; EXCHANGE CONTAINER (LANE 1)
LD 4622.03  ; Flow product number code No.3 (Lane 2)
AND 4620.01  ; EXCHANGE CONTAINER (LANE 2)
ORLD
AND 4623.03  ; Code No.3 fraction workpieces having
ANDNOT 4634.04  ; ...code No.1 fraction workpiece.. taking out
ANDNOT 4634.05  ; ...code No.2 fraction workpiece.. taking out
@AND H160.05  ; 11ST_STEP 05
OR 4634.06  ; ...code No.3 fraction workpiece.. taking out
AND 4634.03  ; Selection of number at taking out positions of fraction workpiece
OUT 4634.06  ; ...code No.3 fraction workpiece.. taking out
; rung 91
LD 4621.04  ; Flow product number code No.4 (Lane 1)
AND 4620.00  ; EXCHANGE CONTAINER (LANE 1)
LD 4622.04  ; Flow product number code No.4 (Lane 2)
AND 4620.01  ; EXCHANGE CONTAINER (LANE 2)
ORLD
AND 4623.04  ; Code No.4 fraction workpieces having
ANDNOT 4634.04  ; ...code No.1 fraction workpiece.. taking out
ANDNOT 4634.05  ; ...code No.2 fraction workpiece.. taking out
ANDNOT 4634.06  ; ...code No.3 fraction workpiece.. taking out
@AND H160.05  ; 11ST_STEP 05
OR 4634.07  ; ...code No.4 fraction workpiece.. taking out
AND 4634.03  ; Selection of number at taking out positions of fraction workpiece
OUT 4634.07  ; ...code No.4 fraction workpiece.. taking out

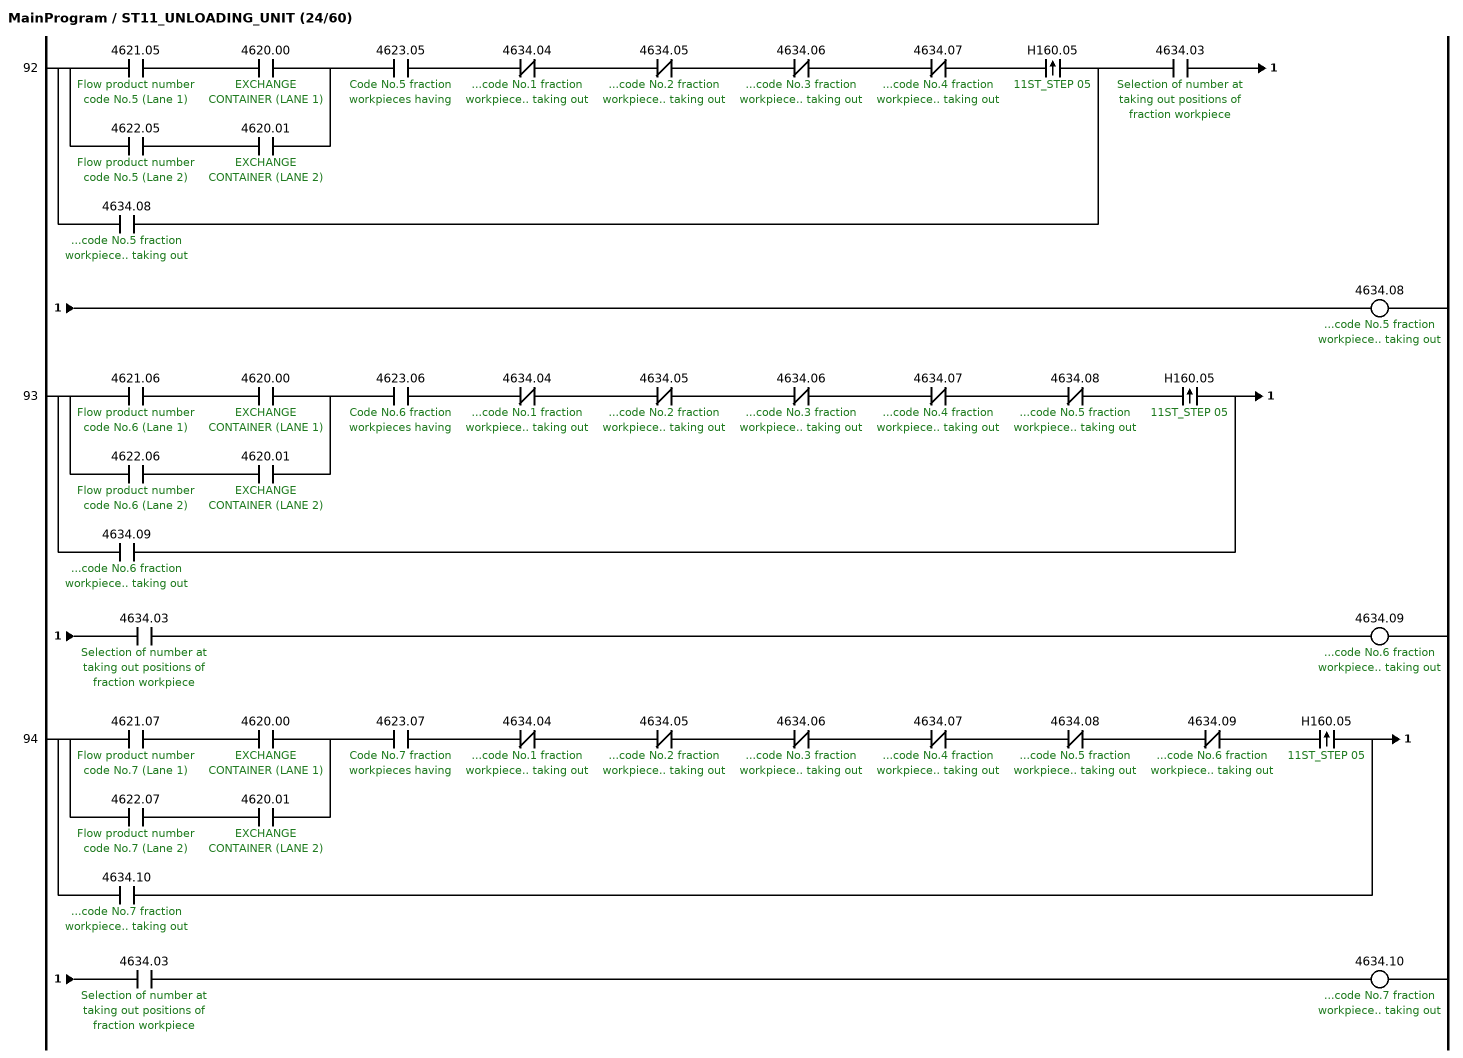
; rung 92
LD 4621.05  ; Flow product number code No.5 (Lane 1)
AND 4620.00  ; EXCHANGE CONTAINER (LANE 1)
LD 4622.05  ; Flow product number code No.5 (Lane 2)
AND 4620.01  ; EXCHANGE CONTAINER (LANE 2)
ORLD
AND 4623.05  ; Code No.5 fraction workpieces having
ANDNOT 4634.04  ; ...code No.1 fraction workpiece.. taking out
ANDNOT 4634.05  ; ...code No.2 fraction workpiece.. taking out
ANDNOT 4634.06  ; ...code No.3 fraction workpiece.. taking out
ANDNOT 4634.07  ; ...code No.4 fraction workpiece.. taking out
@AND H160.05  ; 11ST_STEP 05
OR 4634.08  ; ...code No.5 fraction workpiece.. taking out
AND 4634.03  ; Selection of number at taking out positions of fraction workpiece
OUT 4634.08  ; ...code No.5 fraction workpiece.. taking out
; rung 93
LD 4621.06  ; Flow product number code No.6 (Lane 1)
AND 4620.00  ; EXCHANGE CONTAINER (LANE 1)
LD 4622.06  ; Flow product number code No.6 (Lane 2)
AND 4620.01  ; EXCHANGE CONTAINER (LANE 2)
ORLD
AND 4623.06  ; Code No.6 fraction workpieces having
ANDNOT 4634.04  ; ...code No.1 fraction workpiece.. taking out
ANDNOT 4634.05  ; ...code No.2 fraction workpiece.. taking out
ANDNOT 4634.06  ; ...code No.3 fraction workpiece.. taking out
ANDNOT 4634.07  ; ...code No.4 fraction workpiece.. taking out
ANDNOT 4634.08  ; ...code No.5 fraction workpiece.. taking out
@AND H160.05  ; 11ST_STEP 05
OR 4634.09  ; ...code No.6 fraction workpiece.. taking out
AND 4634.03  ; Selection of number at taking out positions of fraction workpiece
OUT 4634.09  ; ...code No.6 fraction workpiece.. taking out
; rung 94
LD 4621.07  ; Flow product number code No.7 (Lane 1)
AND 4620.00  ; EXCHANGE CONTAINER (LANE 1)
LD 4622.07  ; Flow product number code No.7 (Lane 2)
AND 4620.01  ; EXCHANGE CONTAINER (LANE 2)
ORLD
AND 4623.07  ; Code No.7 fraction workpieces having
ANDNOT 4634.04  ; ...code No.1 fraction workpiece.. taking out
ANDNOT 4634.05  ; ...code No.2 fraction workpiece.. taking out
ANDNOT 4634.06  ; ...code No.3 fraction workpiece.. taking out
ANDNOT 4634.07  ; ...code No.4 fraction workpiece.. taking out
ANDNOT 4634.08  ; ...code No.5 fraction workpiece.. taking out
ANDNOT 4634.09  ; ...code No.6 fraction workpiece.. taking out
@AND H160.05  ; 11ST_STEP 05
OR 4634.10  ; ...code No.7 fraction workpiece.. taking out
AND 4634.03  ; Selection of number at taking out positions of fraction workpiece
OUT 4634.10  ; ...code No.7 fraction workpiece.. taking out

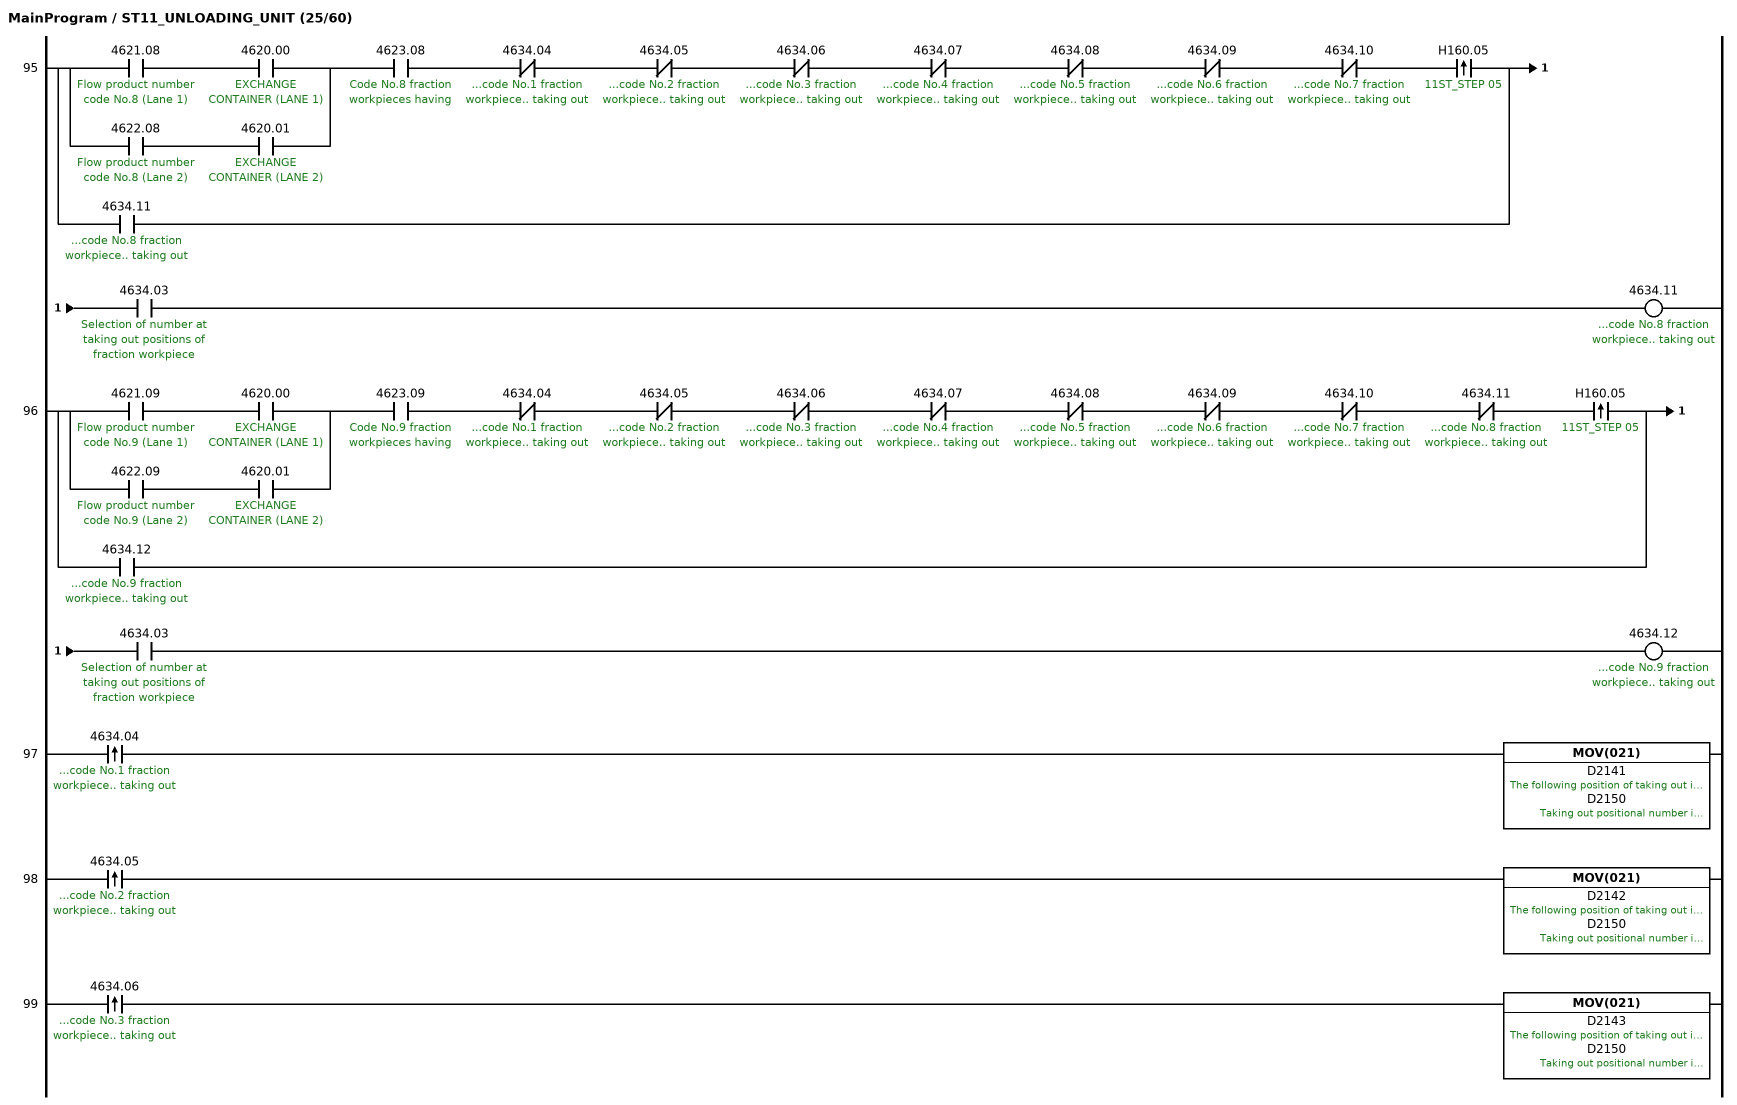
; rung 95
LD 4621.08  ; Flow product number code No.8 (Lane 1)
AND 4620.00  ; EXCHANGE CONTAINER (LANE 1)
LD 4622.08  ; Flow product number code No.8 (Lane 2)
AND 4620.01  ; EXCHANGE CONTAINER (LANE 2)
ORLD
AND 4623.08  ; Code No.8 fraction workpieces having
ANDNOT 4634.04  ; ...code No.1 fraction workpiece.. taking out
ANDNOT 4634.05  ; ...code No.2 fraction workpiece.. taking out
ANDNOT 4634.06  ; ...code No.3 fraction workpiece.. taking out
ANDNOT 4634.07  ; ...code No.4 fraction workpiece.. taking out
ANDNOT 4634.08  ; ...code No.5 fraction workpiece.. taking out
ANDNOT 4634.09  ; ...code No.6 fraction workpiece.. taking out
ANDNOT 4634.10  ; ...code No.7 fraction workpiece.. taking out
@AND H160.05  ; 11ST_STEP 05
OR 4634.11  ; ...code No.8 fraction workpiece.. taking out
AND 4634.03  ; Selection of number at taking out positions of fraction workpiece
OUT 4634.11  ; ...code No.8 fraction workpiece.. taking out
; rung 96
LD 4621.09  ; Flow product number code No.9 (Lane 1)
AND 4620.00  ; EXCHANGE CONTAINER (LANE 1)
LD 4622.09  ; Flow product number code No.9 (Lane 2)
AND 4620.01  ; EXCHANGE CONTAINER (LANE 2)
ORLD
AND 4623.09  ; Code No.9 fraction workpieces having
ANDNOT 4634.04  ; ...code No.1 fraction workpiece.. taking out
ANDNOT 4634.05  ; ...code No.2 fraction workpiece.. taking out
ANDNOT 4634.06  ; ...code No.3 fraction workpiece.. taking out
ANDNOT 4634.07  ; ...code No.4 fraction workpiece.. taking out
ANDNOT 4634.08  ; ...code No.5 fraction workpiece.. taking out
ANDNOT 4634.09  ; ...code No.6 fraction workpiece.. taking out
ANDNOT 4634.10  ; ...code No.7 fraction workpiece.. taking out
ANDNOT 4634.11  ; ...code No.8 fraction workpiece.. taking out
@AND H160.05  ; 11ST_STEP 05
OR 4634.12  ; ...code No.9 fraction workpiece.. taking out
AND 4634.03  ; Selection of number at taking out positions of fraction workpiece
OUT 4634.12  ; ...code No.9 fraction workpiece.. taking out
; rung 97
@LD 4634.04  ; ...code No.1 fraction workpiece.. taking out
MOV(021) D2141 D2150  ; The following position of taking out in a container number in fraction workpiece (code no.1), Taking out positional number in fraction workpiece
; rung 98
@LD 4634.05  ; ...code No.2 fraction workpiece.. taking out
MOV(021) D2142 D2150  ; The following position of taking out in a container number in fraction workpiece (code no.2), Taking out positional number in fraction workpiece
; rung 99
@LD 4634.06  ; ...code No.3 fraction workpiece.. taking out
MOV(021) D2143 D2150  ; The following position of taking out in a container number in fraction workpiece (code no.3), Taking out positional number in fraction workpiece

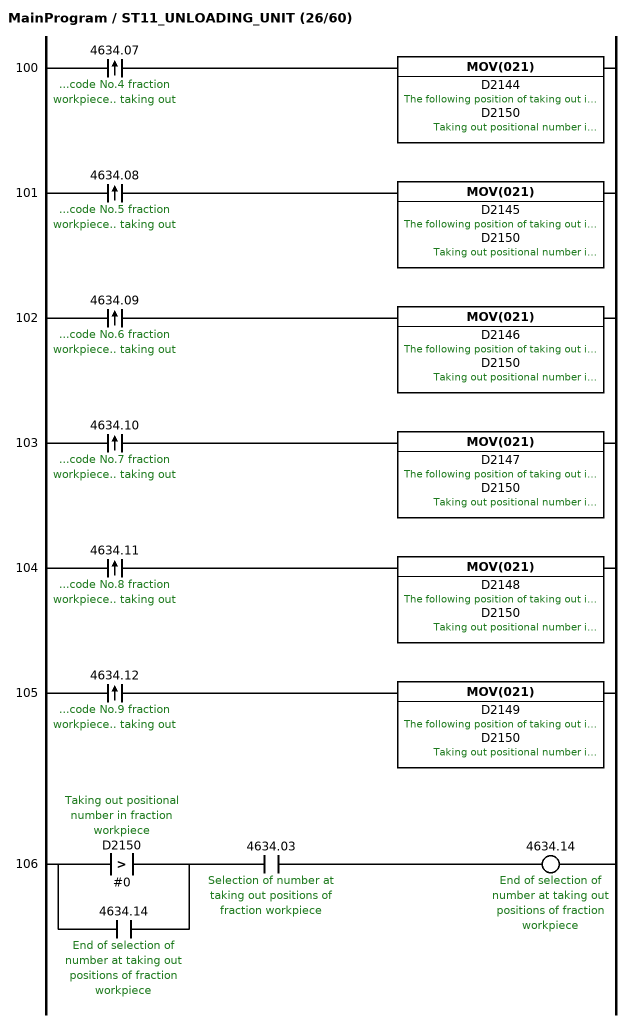
; rung 100
@LD 4634.07  ; ...code No.4 fraction workpiece.. taking out
MOV(021) D2144 D2150  ; The following position of taking out in a container number in fraction workpiece (code no.4), Taking out positional number in fraction workpiece
; rung 101
@LD 4634.08  ; ...code No.5 fraction workpiece.. taking out
MOV(021) D2145 D2150  ; The following position of taking out in a container number in fraction workpiece (code no.5), Taking out positional number in fraction workpiece
; rung 102
@LD 4634.09  ; ...code No.6 fraction workpiece.. taking out
MOV(021) D2146 D2150  ; The following position of taking out in a container number in fraction workpiece (code no.6), Taking out positional number in fraction workpiece
; rung 103
@LD 4634.10  ; ...code No.7 fraction workpiece.. taking out
MOV(021) D2147 D2150  ; The following position of taking out in a container number in fraction workpiece (code no.7), Taking out positional number in fraction workpiece
; rung 104
@LD 4634.11  ; ...code No.8 fraction workpiece.. taking out
MOV(021) D2148 D2150  ; The following position of taking out in a container number in fraction workpiece (code no.8), Taking out positional number in fraction workpiece
; rung 105
@LD 4634.12  ; ...code No.9 fraction workpiece.. taking out
MOV(021) D2149 D2150  ; The following position of taking out in a container number in fraction workpiece (code no.9), Taking out positional number in fraction workpiece
; rung 106
LD>(320) D2150 #0  ; Taking out positional number in fraction workpiece
OR 4634.14  ; End of selection of number at taking out positions of fraction workpiece
AND 4634.03  ; Selection of number at taking out positions of fraction workpiece
OUT 4634.14  ; End of selection of number at taking out positions of fraction workpiece

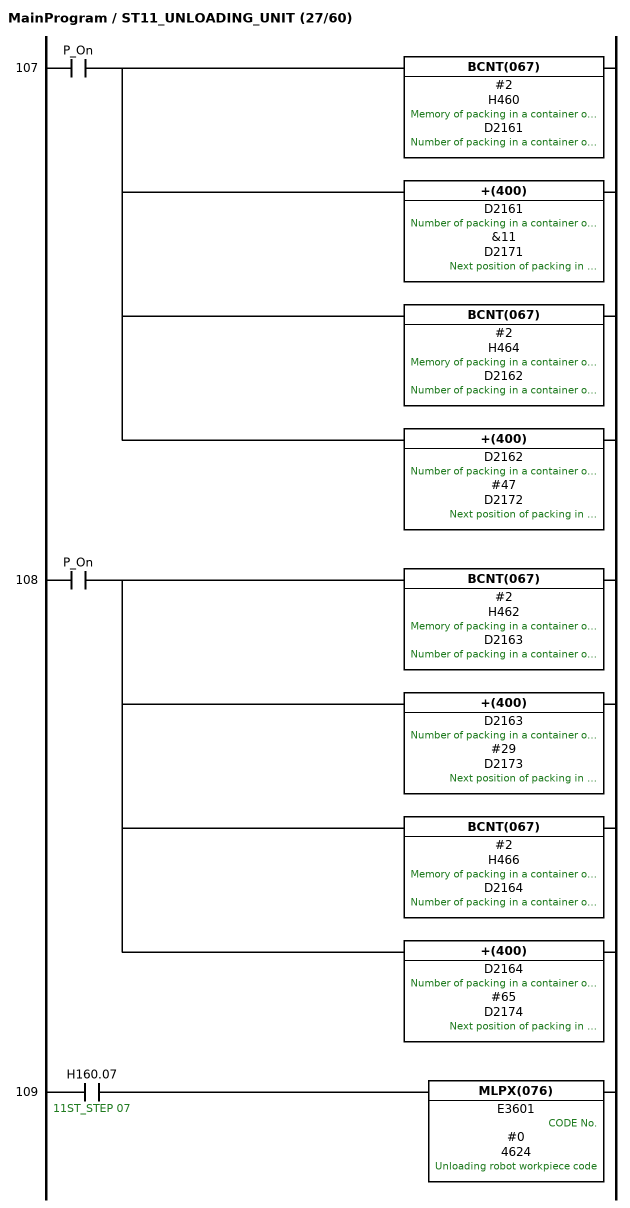
; rung 107
LD P_On
BCNT(067) #2 H460 D2161  ; Memory of packing in a container of lane 1 (exchange container), Number of packing in a container of lane 1 (exchange container)(BIN)
+(400) D2161 &11 D2171  ; Number of packing in a container of lane 1 (exchange container)(BIN), Next position of packing in a container of lane 1 (exchange container)(BIN)
BCNT(067) #2 H464 D2162  ; Memory of packing in a container of lane 2 (exchange container), Number of packing in a container of lane 2 (exchange container)(BIN)
+(400) D2162 #47 D2172  ; Number of packing in a container of lane 2 (exchange container)(BIN), Next position of packing in a container of lane 2 (exchange container)(BIN)
; rung 108
LD P_On
BCNT(067) #2 H462 D2163  ; Memory of packing in a container of lane 1 (container befor exchange), Number of packing in a container of lane 1 (container before exchange)(BIN)
+(400) D2163 #29 D2173  ; Number of packing in a container of lane 1 (container before exchange)(BIN), Next position of packing in a container of lane 3 (exchange container)(BIN)
BCNT(067) #2 H466 D2164  ; Memory of packing in a container of lane 2 (container befor exchange), Number of packing in a container of lane 2 (container before exchange)(BIN)
+(400) D2164 #65 D2174  ; Number of packing in a container of lane 2 (container before exchange)(BIN), Next position of packing in a container of lane 4 (exchange container)(BIN)
; rung 109
LD H160.07  ; 11ST_STEP 07
MLPX(076) E3601 #0 4624  ; CODE No., Unloading robot workpiece code

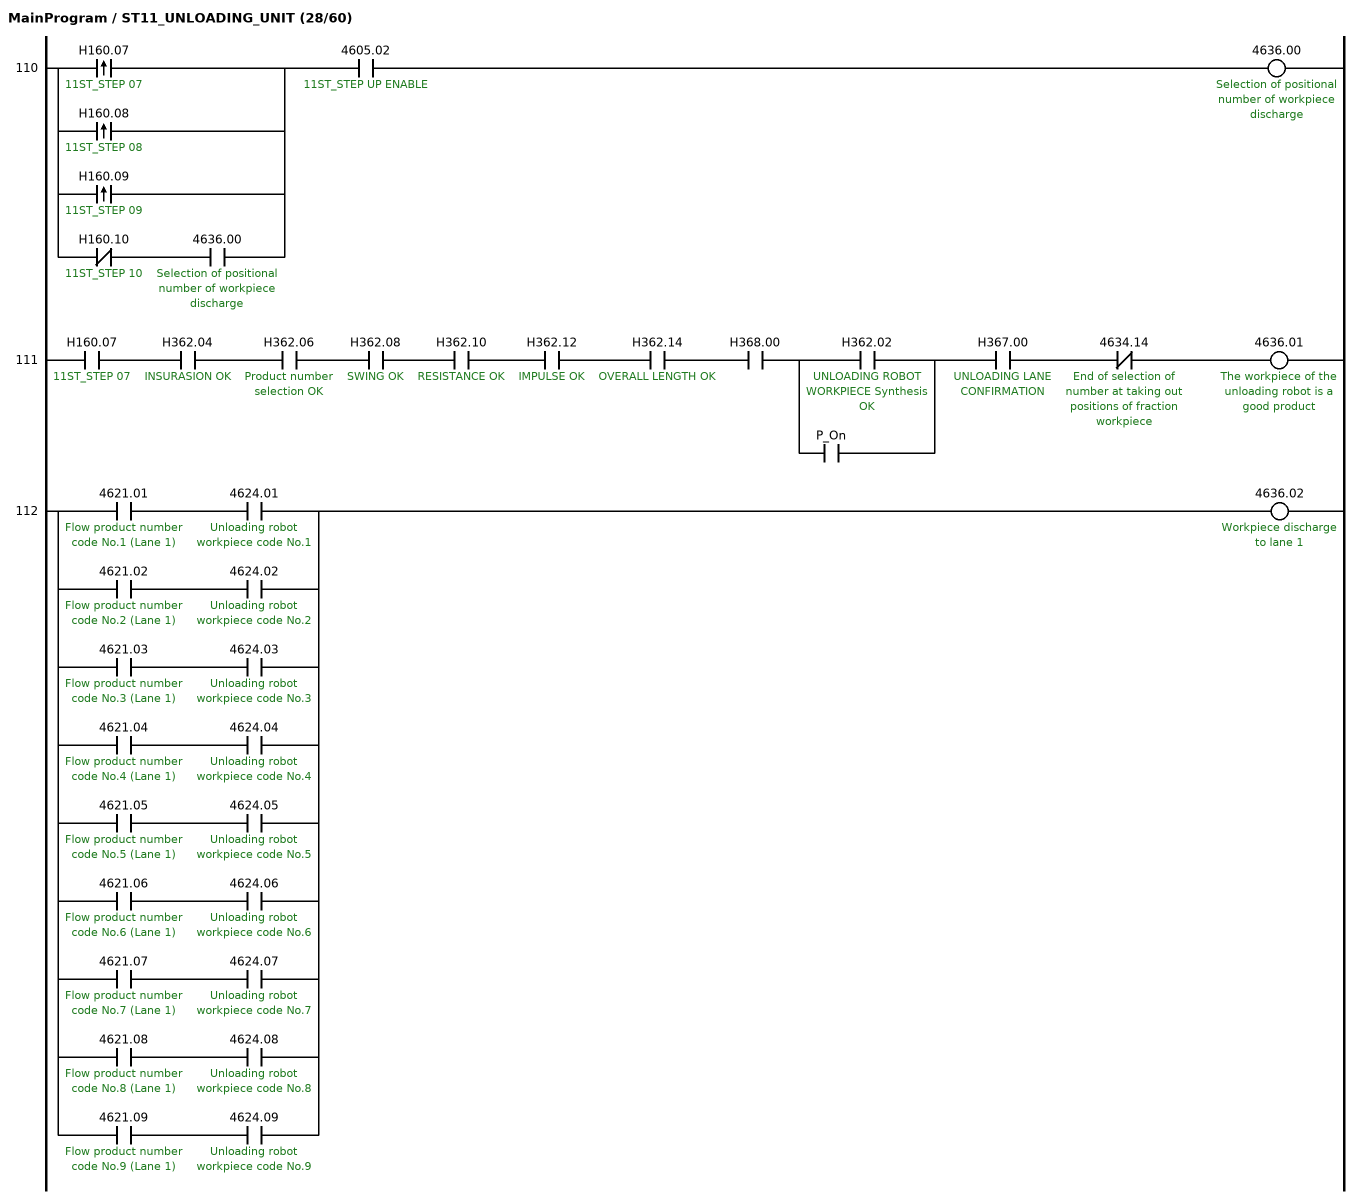
; rung 110
@LD H160.07  ; 11ST_STEP 07
@OR H160.08  ; 11ST_STEP 08
@OR H160.09  ; 11ST_STEP 09
LDNOT H160.10  ; 11ST_STEP 10
AND 4636.00  ; Selection of positional number of workpiece discharge
ORLD
AND 4605.02  ; 11ST_STEP UP ENABLE
OUT 4636.00  ; Selection of positional number of workpiece discharge
; rung 111
LD H160.07  ; 11ST_STEP 07
AND H362.04  ; INSURASION OK
AND H362.06  ; Product number selection OK
AND H362.08  ; SWING OK
AND H362.10  ; RESISTANCE OK
AND H362.12  ; IMPULSE OK
AND H362.14  ; OVERALL LENGTH OK
AND H368.00
LD H362.02  ; UNLOADING ROBOT WORKPIECE Synthesis OK
OR P_On
ANDLD
AND H367.00  ; UNLOADING LANE CONFIRMATION
ANDNOT 4634.14  ; End of selection of number at taking out positions of fraction workpiece
OUT 4636.01  ; The workpiece of the unloading robot is a good product
; rung 112
LD 4621.01  ; Flow product number code No.1 (Lane 1)
AND 4624.01  ; Unloading robot workpiece code No.1
LD 4621.02  ; Flow product number code No.2 (Lane 1)
AND 4624.02  ; Unloading robot workpiece code No.2
ORLD
LD 4621.03  ; Flow product number code No.3 (Lane 1)
AND 4624.03  ; Unloading robot workpiece code No.3
ORLD
LD 4621.04  ; Flow product number code No.4 (Lane 1)
AND 4624.04  ; Unloading robot workpiece code No.4
ORLD
LD 4621.05  ; Flow product number code No.5 (Lane 1)
AND 4624.05  ; Unloading robot workpiece code No.5
ORLD
LD 4621.06  ; Flow product number code No.6 (Lane 1)
AND 4624.06  ; Unloading robot workpiece code No.6
ORLD
LD 4621.07  ; Flow product number code No.7 (Lane 1)
AND 4624.07  ; Unloading robot workpiece code No.7
ORLD
LD 4621.08  ; Flow product number code No.8 (Lane 1)
AND 4624.08  ; Unloading robot workpiece code No.8
ORLD
LD 4621.09  ; Flow product number code No.9 (Lane 1)
AND 4624.09  ; Unloading robot workpiece code No.9
ORLD
OUT 4636.02  ; Workpiece discharge to lane 1

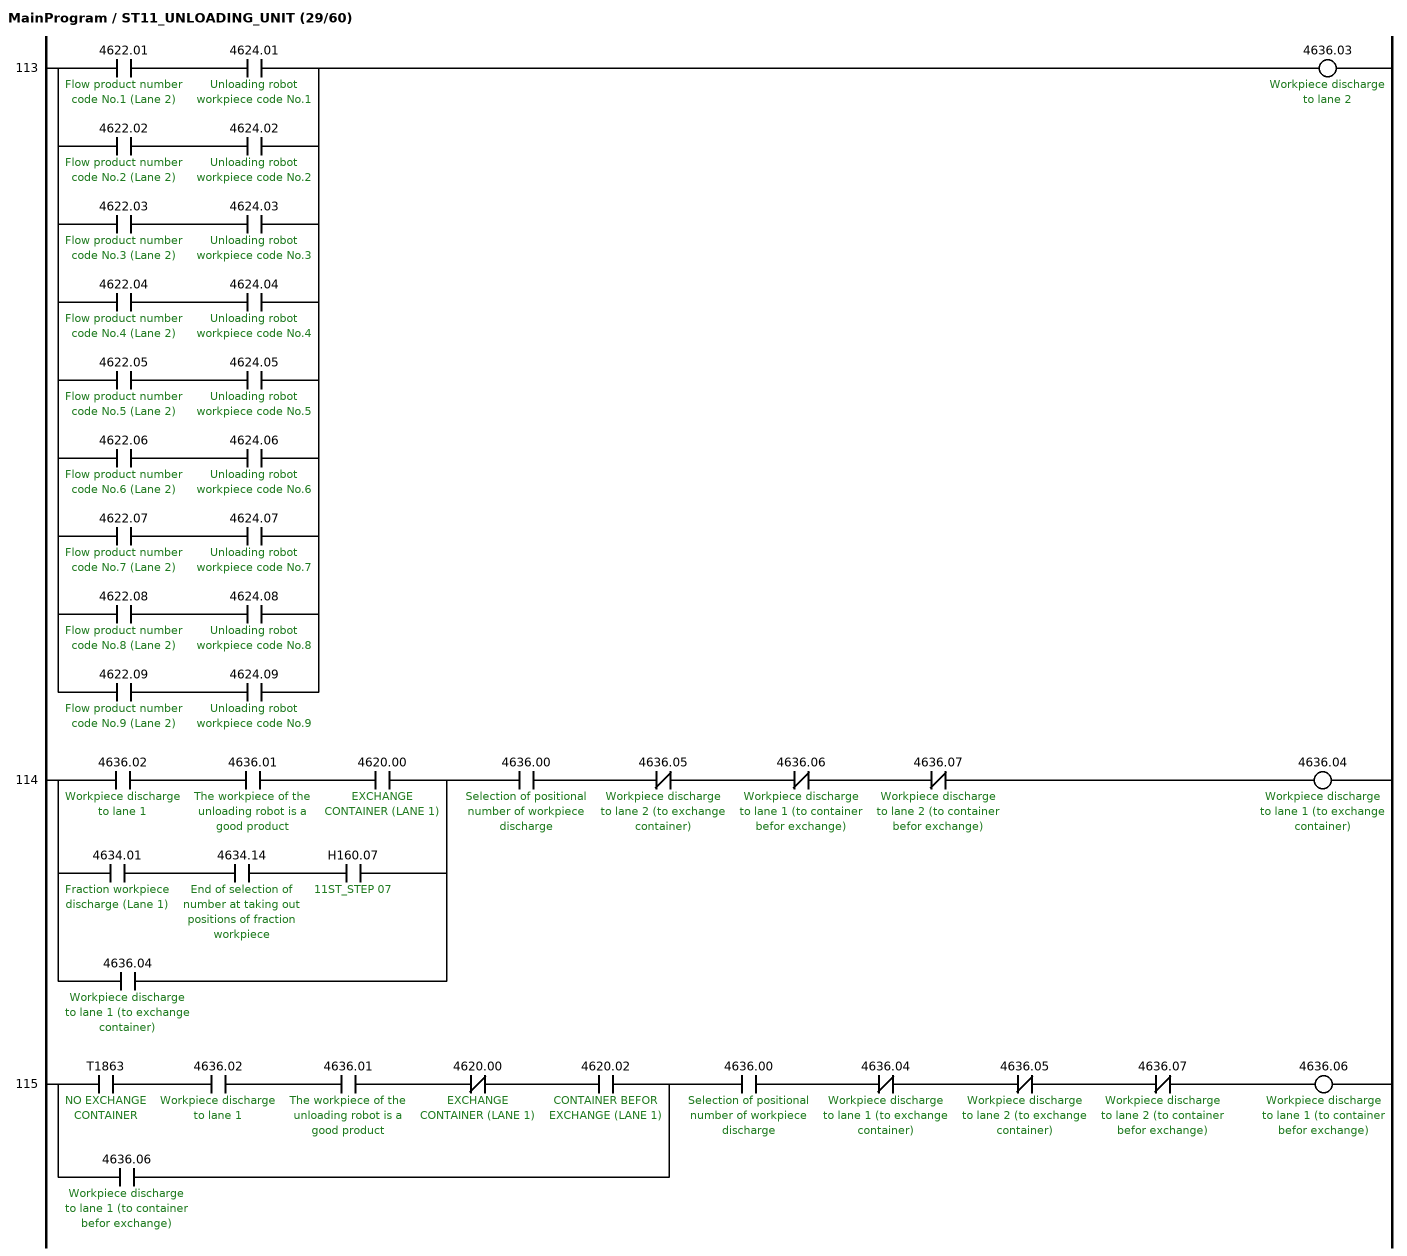
; rung 113
LD 4622.01  ; Flow product number code No.1 (Lane 2)
AND 4624.01  ; Unloading robot workpiece code No.1
LD 4622.02  ; Flow product number code No.2 (Lane 2)
AND 4624.02  ; Unloading robot workpiece code No.2
ORLD
LD 4622.03  ; Flow product number code No.3 (Lane 2)
AND 4624.03  ; Unloading robot workpiece code No.3
ORLD
LD 4622.04  ; Flow product number code No.4 (Lane 2)
AND 4624.04  ; Unloading robot workpiece code No.4
ORLD
LD 4622.05  ; Flow product number code No.5 (Lane 2)
AND 4624.05  ; Unloading robot workpiece code No.5
ORLD
LD 4622.06  ; Flow product number code No.6 (Lane 2)
AND 4624.06  ; Unloading robot workpiece code No.6
ORLD
LD 4622.07  ; Flow product number code No.7 (Lane 2)
AND 4624.07  ; Unloading robot workpiece code No.7
ORLD
LD 4622.08  ; Flow product number code No.8 (Lane 2)
AND 4624.08  ; Unloading robot workpiece code No.8
ORLD
LD 4622.09  ; Flow product number code No.9 (Lane 2)
AND 4624.09  ; Unloading robot workpiece code No.9
ORLD
OUT 4636.03  ; Workpiece discharge to lane 2
; rung 114
LD 4636.02  ; Workpiece discharge to lane 1
AND 4636.01  ; The workpiece of the unloading robot is a good product
AND 4620.00  ; EXCHANGE CONTAINER (LANE 1)
LD 4634.01  ; Fraction workpiece discharge (Lane 1)
AND 4634.14  ; End of selection of number at taking out positions of fraction workpiece
AND H160.07  ; 11ST_STEP 07
ORLD
OR 4636.04  ; Workpiece discharge to lane 1 (to exchange container)
AND 4636.00  ; Selection of positional number of workpiece discharge
ANDNOT 4636.05  ; Workpiece discharge to lane 2 (to exchange container)
ANDNOT 4636.06  ; Workpiece discharge to lane 1 (to container befor exchange)
ANDNOT 4636.07  ; Workpiece discharge to lane 2 (to container befor exchange)
OUT 4636.04  ; Workpiece discharge to lane 1 (to exchange container)
; rung 115
LD T1863  ; NO EXCHANGE CONTAINER
AND 4636.02  ; Workpiece discharge to lane 1
AND 4636.01  ; The workpiece of the unloading robot is a good product
ANDNOT 4620.00  ; EXCHANGE CONTAINER (LANE 1)
AND 4620.02  ; CONTAINER BEFOR EXCHANGE (LANE 1)
OR 4636.06  ; Workpiece discharge to lane 1 (to container befor exchange)
AND 4636.00  ; Selection of positional number of workpiece discharge
ANDNOT 4636.04  ; Workpiece discharge to lane 1 (to exchange container)
ANDNOT 4636.05  ; Workpiece discharge to lane 2 (to exchange container)
ANDNOT 4636.07  ; Workpiece discharge to lane 2 (to container befor exchange)
OUT 4636.06  ; Workpiece discharge to lane 1 (to container befor exchange)

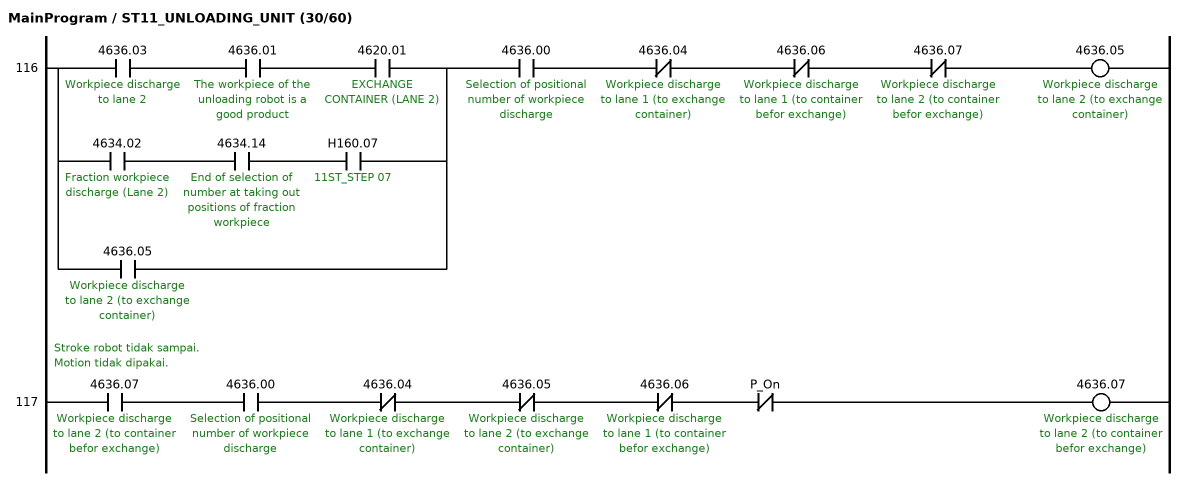
; rung 116
LD 4636.03  ; Workpiece discharge to lane 2
AND 4636.01  ; The workpiece of the unloading robot is a good product
AND 4620.01  ; EXCHANGE CONTAINER (LANE 2)
LD 4634.02  ; Fraction workpiece discharge (Lane 2)
AND 4634.14  ; End of selection of number at taking out positions of fraction workpiece
AND H160.07  ; 11ST_STEP 07
ORLD
OR 4636.05  ; Workpiece discharge to lane 2 (to exchange container)
AND 4636.00  ; Selection of positional number of workpiece discharge
ANDNOT 4636.04  ; Workpiece discharge to lane 1 (to exchange container)
ANDNOT 4636.06  ; Workpiece discharge to lane 1 (to container befor exchange)
ANDNOT 4636.07  ; Workpiece discharge to lane 2 (to container befor exchange)
OUT 4636.05  ; Workpiece discharge to lane 2 (to exchange container)
; rung 117: Stroke robot tidak sampai. / Motion tidak dipakai.
LD 4636.07  ; Workpiece discharge to lane 2 (to container befor exchange)
AND 4636.00  ; Selection of positional number of workpiece discharge
ANDNOT 4636.04  ; Workpiece discharge to lane 1 (to exchange container)
ANDNOT 4636.05  ; Workpiece discharge to lane 2 (to exchange container)
ANDNOT 4636.06  ; Workpiece discharge to lane 1 (to container befor exchange)
ANDNOT P_On
OUT 4636.07  ; Workpiece discharge to lane 2 (to container befor exchange)

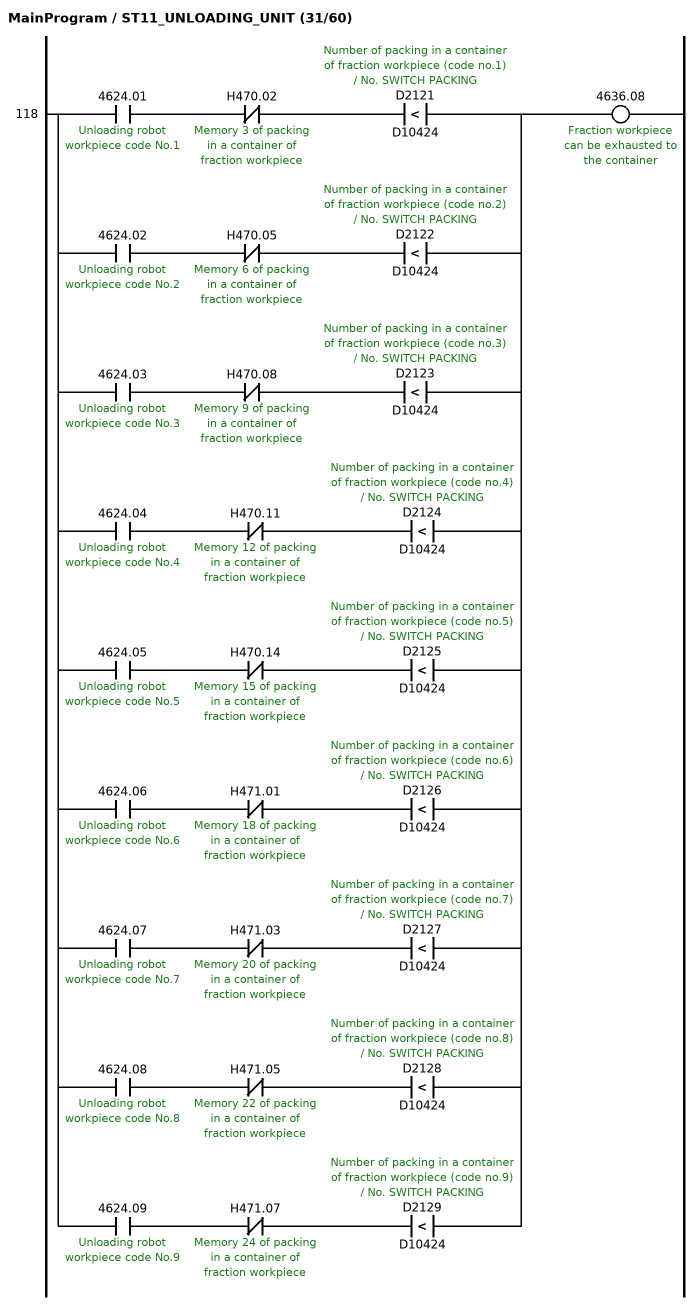
; rung 118
LD 4624.01  ; Unloading robot workpiece code No.1
ANDNOT H470.02  ; Memory 3 of packing in a container of fraction workpiece
AND<(310) D2121 D10424  ; Number of packing in a container of fraction workpiece (code no.1), No. SWITCH PACKING
LD 4624.02  ; Unloading robot workpiece code No.2
ANDNOT H470.05  ; Memory 6 of packing in a container of fraction workpiece
AND<(310) D2122 D10424  ; Number of packing in a container of fraction workpiece (code no.2), No. SWITCH PACKING
ORLD
LD 4624.03  ; Unloading robot workpiece code No.3
ANDNOT H470.08  ; Memory 9 of packing in a container of fraction workpiece
AND<(310) D2123 D10424  ; Number of packing in a container of fraction workpiece (code no.3), No. SWITCH PACKING
ORLD
LD 4624.04  ; Unloading robot workpiece code No.4
ANDNOT H470.11  ; Memory 12 of packing in a container of fraction workpiece
AND<(310) D2124 D10424  ; Number of packing in a container of fraction workpiece (code no.4), No. SWITCH PACKING
ORLD
LD 4624.05  ; Unloading robot workpiece code No.5
ANDNOT H470.14  ; Memory 15 of packing in a container of fraction workpiece
AND<(310) D2125 D10424  ; Number of packing in a container of fraction workpiece (code no.5), No. SWITCH PACKING
ORLD
LD 4624.06  ; Unloading robot workpiece code No.6
ANDNOT H471.01  ; Memory 18 of packing in a container of fraction workpiece
AND<(310) D2126 D10424  ; Number of packing in a container of fraction workpiece (code no.6), No. SWITCH PACKING
ORLD
LD 4624.07  ; Unloading robot workpiece code No.7
ANDNOT H471.03  ; Memory 20 of packing in a container of fraction workpiece
AND<(310) D2127 D10424  ; Number of packing in a container of fraction workpiece (code no.7), No. SWITCH PACKING
ORLD
LD 4624.08  ; Unloading robot workpiece code No.8
ANDNOT H471.05  ; Memory 22 of packing in a container of fraction workpiece
AND<(310) D2128 D10424  ; Number of packing in a container of fraction workpiece (code no.8), No. SWITCH PACKING
ORLD
LD 4624.09  ; Unloading robot workpiece code No.9
ANDNOT H471.07  ; Memory 24 of packing in a container of fraction workpiece
AND<(310) D2129 D10424  ; Number of packing in a container of fraction workpiece (code no.9), No. SWITCH PACKING
ORLD
OUT 4636.08  ; Fraction workpiece can be exhausted to the container

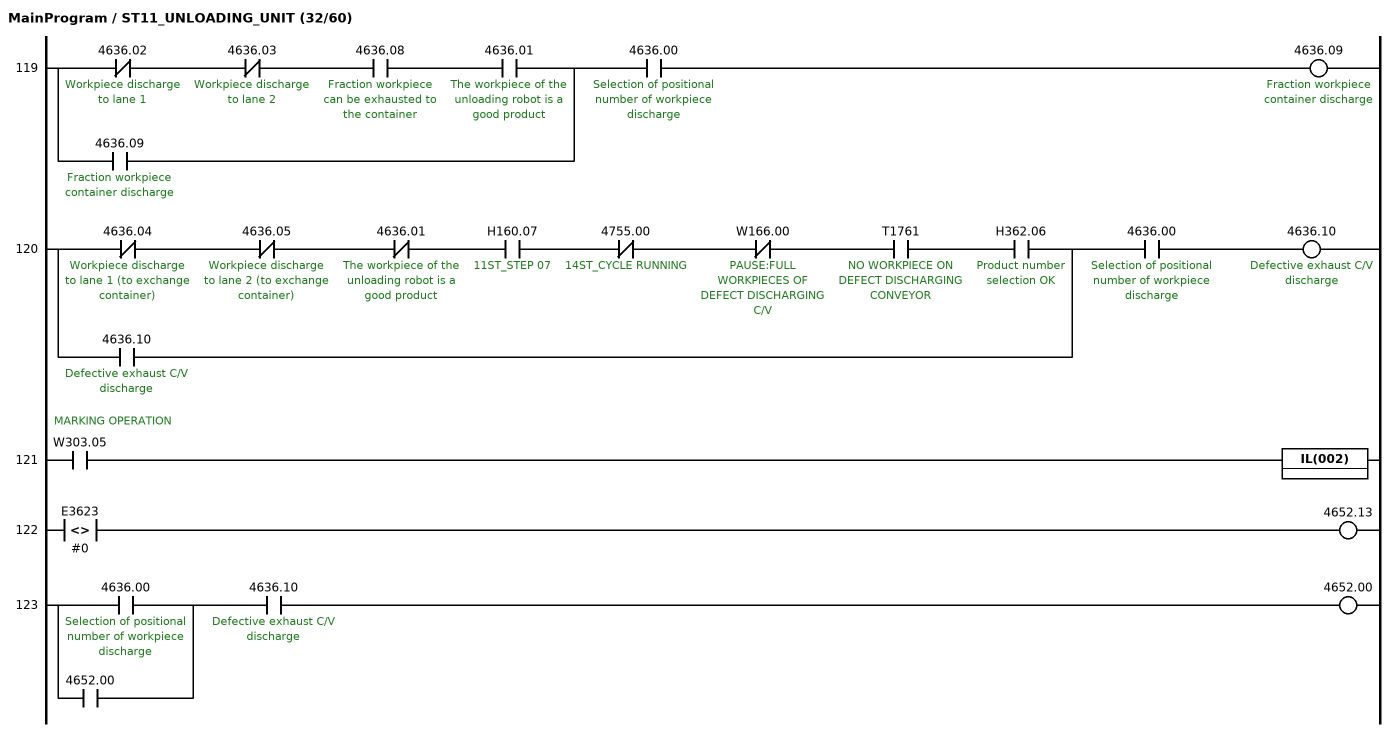
; rung 119
LDNOT 4636.02  ; Workpiece discharge to lane 1
ANDNOT 4636.03  ; Workpiece discharge to lane 2
AND 4636.08  ; Fraction workpiece can be exhausted to the container
AND 4636.01  ; The workpiece of the unloading robot is a good product
OR 4636.09  ; Fraction workpiece container discharge
AND 4636.00  ; Selection of positional number of workpiece discharge
OUT 4636.09  ; Fraction workpiece container discharge
; rung 120
LDNOT 4636.04  ; Workpiece discharge to lane 1 (to exchange container)
ANDNOT 4636.05  ; Workpiece discharge to lane 2 (to exchange container)
ANDNOT 4636.01  ; The workpiece of the unloading robot is a good product
AND H160.07  ; 11ST_STEP 07
ANDNOT 4755.00  ; 14ST_CYCLE RUNNING
ANDNOT W166.00  ; PAUSE:FULL WORKPIECES OF DEFECT DISCHARGING C/V
AND T1761  ; NO WORKPIECE ON DEFECT DISCHARGING CONVEYOR
AND H362.06  ; Product number selection OK
OR 4636.10  ; Defective exhaust C/V discharge
AND 4636.00  ; Selection of positional number of workpiece discharge
OUT 4636.10  ; Defective exhaust C/V discharge
; rung 121: MARKING OPERATION
LD W303.05
IL(002)
; rung 122
LD<>(305) E3623 #0
OUT 4652.13
; rung 123
LD 4636.00  ; Selection of positional number of workpiece discharge
OR 4652.00
AND 4636.10  ; Defective exhaust C/V discharge
OUT 4652.00

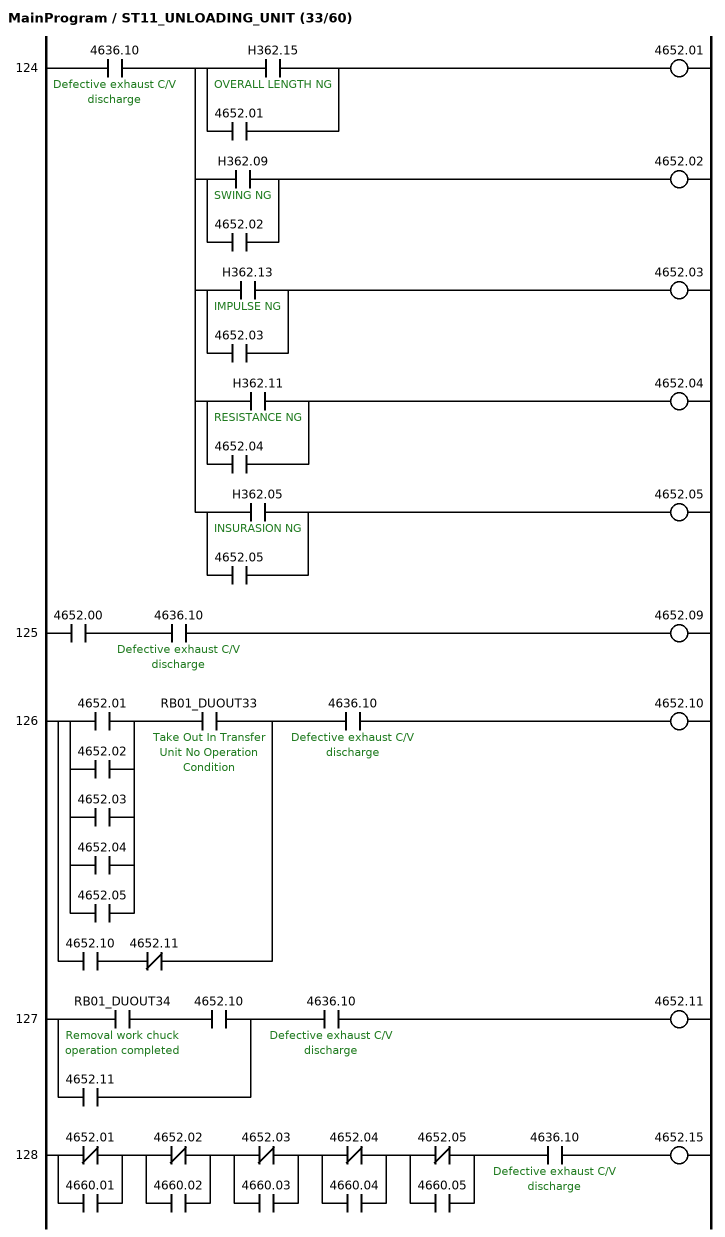
; rung 124
LD 4636.10  ; Defective exhaust C/V discharge
OUT TR0
LD H362.15  ; OVERALL LENGTH NG
OR 4652.01
ANDLD
OUT 4652.01
LD TR0
LD H362.09  ; SWING NG
OR 4652.02
ANDLD
OUT 4652.02
LD TR0
LD H362.13  ; IMPULSE NG
OR 4652.03
ANDLD
OUT 4652.03
LD TR0
LD H362.11  ; RESISTANCE NG
OR 4652.04
ANDLD
OUT 4652.04
LD TR0
LD H362.05  ; INSURASION NG
OR 4652.05
ANDLD
OUT 4652.05
; rung 125
LD 4652.00
AND 4636.10  ; Defective exhaust C/V discharge
OUT 4652.09
; rung 126
LD 4652.01
OR 4652.02
OR 4652.03
OR 4652.04
OR 4652.05
AND RB01_DUOUT33  ; Take Out In Transfer Unit No Operation Condition
LD 4652.10
ANDNOT 4652.11
ORLD
AND 4636.10  ; Defective exhaust C/V discharge
OUT 4652.10
; rung 127
LD RB01_DUOUT34  ; Removal work chuck operation completed
AND 4652.10
OR 4652.11
AND 4636.10  ; Defective exhaust C/V discharge
OUT 4652.11
; rung 128
LDNOT 4652.01
OR 4660.01
LDNOT 4652.02
OR 4660.02
ANDLD
LDNOT 4652.03
OR 4660.03
ANDLD
LDNOT 4652.04
OR 4660.04
ANDLD
LDNOT 4652.05
OR 4660.05
ANDLD
AND 4636.10  ; Defective exhaust C/V discharge
OUT 4652.15

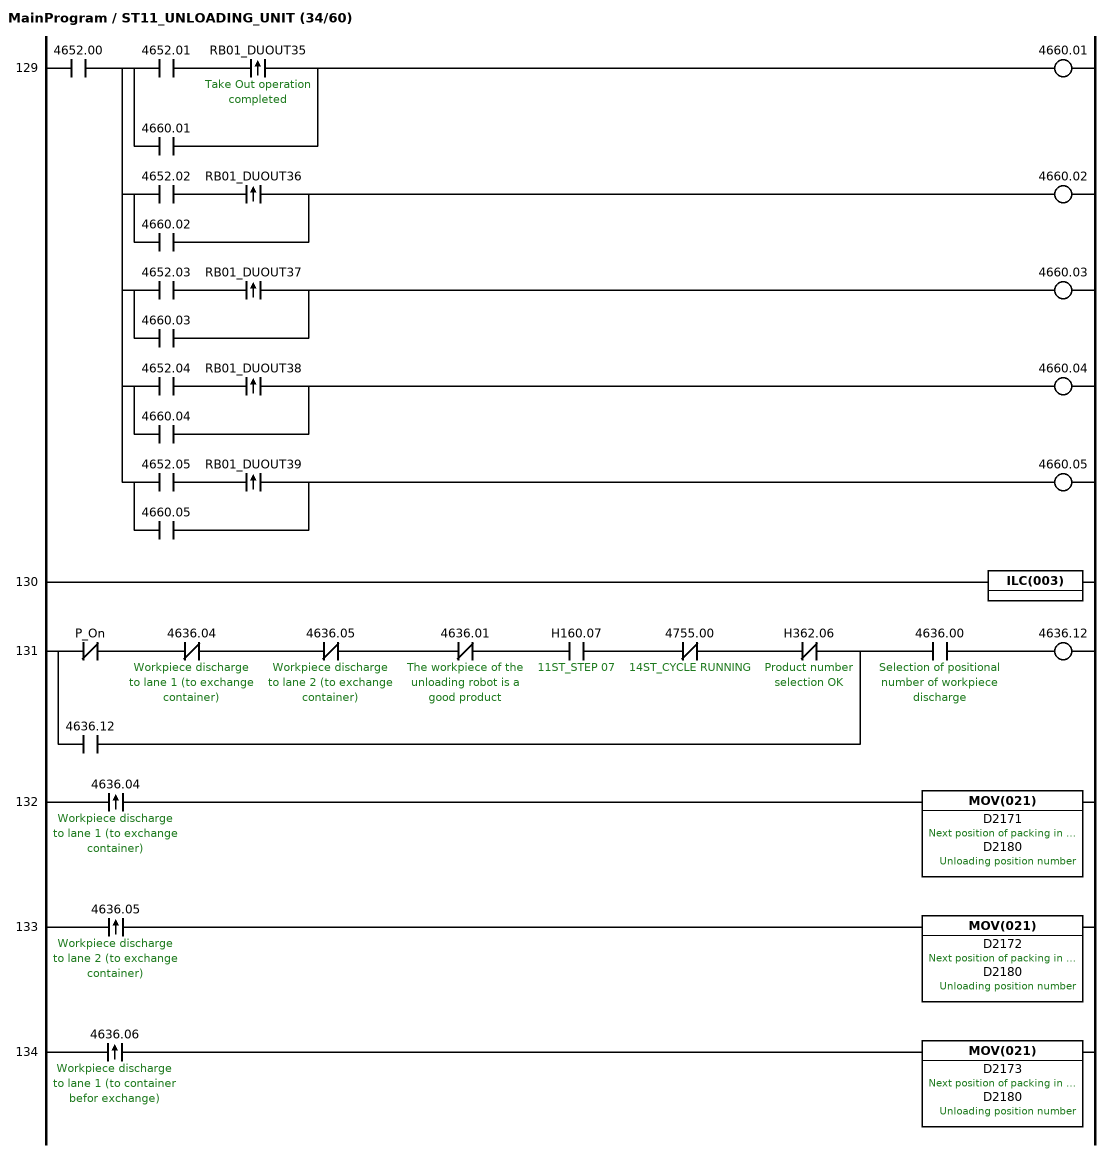
; rung 129
LD 4652.00
OUT TR0
LD 4652.01
@AND RB01_DUOUT35  ; Take Out operation completed
OR 4660.01
ANDLD
OUT 4660.01
LD TR0
LD 4652.02
@AND RB01_DUOUT36
OR 4660.02
ANDLD
OUT 4660.02
LD TR0
LD 4652.03
@AND RB01_DUOUT37
OR 4660.03
ANDLD
OUT 4660.03
LD TR0
LD 4652.04
@AND RB01_DUOUT38
OR 4660.04
ANDLD
OUT 4660.04
LD TR0
LD 4652.05
@AND RB01_DUOUT39
OR 4660.05
ANDLD
OUT 4660.05
; rung 130
ILC(003)
; rung 131
LDNOT P_On
ANDNOT 4636.04  ; Workpiece discharge to lane 1 (to exchange container)
ANDNOT 4636.05  ; Workpiece discharge to lane 2 (to exchange container)
ANDNOT 4636.01  ; The workpiece of the unloading robot is a good product
AND H160.07  ; 11ST_STEP 07
ANDNOT 4755.00  ; 14ST_CYCLE RUNNING
ANDNOT H362.06  ; Product number selection OK
OR 4636.12
AND 4636.00  ; Selection of positional number of workpiece discharge
OUT 4636.12
; rung 132
@LD 4636.04  ; Workpiece discharge to lane 1 (to exchange container)
MOV(021) D2171 D2180  ; Next position of packing in a container of lane 1 (exchange container)(BIN), Unloading position number
; rung 133
@LD 4636.05  ; Workpiece discharge to lane 2 (to exchange container)
MOV(021) D2172 D2180  ; Next position of packing in a container of lane 2 (exchange container)(BIN), Unloading position number
; rung 134
@LD 4636.06  ; Workpiece discharge to lane 1 (to container befor exchange)
MOV(021) D2173 D2180  ; Next position of packing in a container of lane 3 (exchange container)(BIN), Unloading position number

